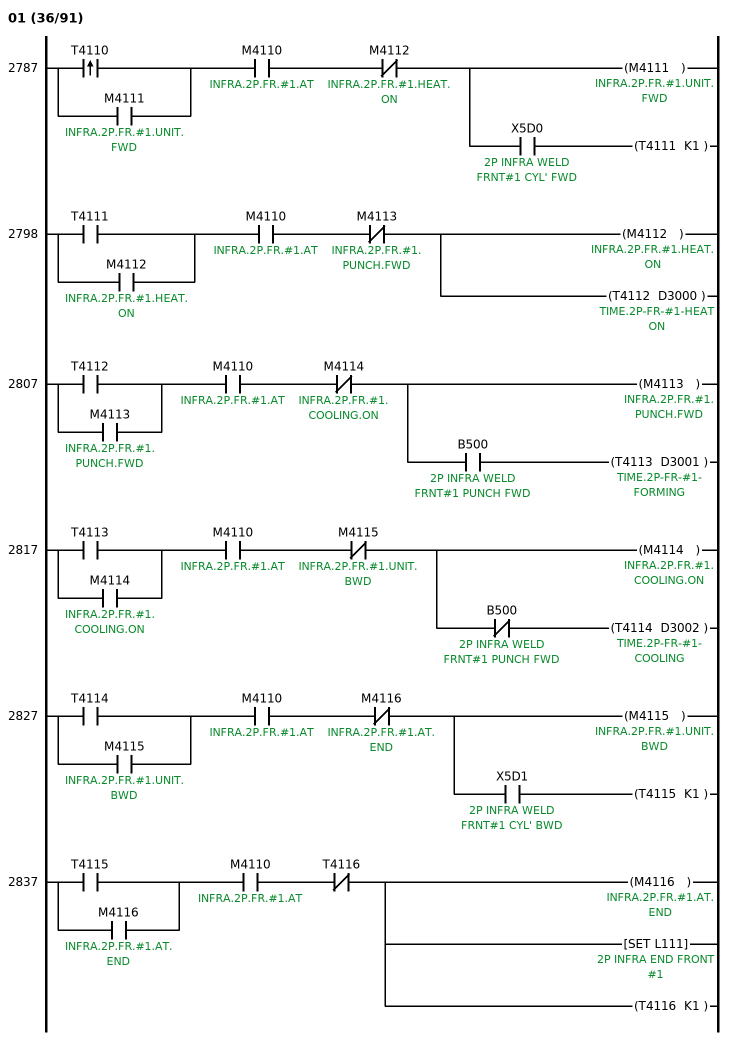
2787  LDP     T4110
      OR      M4111  ; INFRA.2P.FR.#1.UNIT.FWD
      AND     M4110  ; INFRA.2P.FR.#1.AT
      ANI     M4112  ; INFRA.2P.FR.#1.HEAT.ON
      OUT     M4111  ; INFRA.2P.FR.#1.UNIT.FWD
      AND     X5D0  ; 2P INFRA WELD FRNT#1 CYL' FWD
      OUT     T4111 K1
2798  LD      T4111
      OR      M4112  ; INFRA.2P.FR.#1.HEAT.ON
      AND     M4110  ; INFRA.2P.FR.#1.AT
      ANI     M4113  ; INFRA.2P.FR.#1.PUNCH.FWD
      OUT     M4112  ; INFRA.2P.FR.#1.HEAT.ON
      OUT     T4112 D3000  ; TIME.2P-FR-#1-HEAT ON
2807  LD      T4112
      OR      M4113  ; INFRA.2P.FR.#1.PUNCH.FWD
      AND     M4110  ; INFRA.2P.FR.#1.AT
      ANI     M4114  ; INFRA.2P.FR.#1.COOLING.ON
      OUT     M4113  ; INFRA.2P.FR.#1.PUNCH.FWD
      AND     B500  ; 2P INFRA WELD FRNT#1 PUNCH FWD
      OUT     T4113 D3001  ; TIME.2P-FR-#1-FORMING
2817  LD      T4113
      OR      M4114  ; INFRA.2P.FR.#1.COOLING.ON
      AND     M4110  ; INFRA.2P.FR.#1.AT
      ANI     M4115  ; INFRA.2P.FR.#1.UNIT.BWD
      OUT     M4114  ; INFRA.2P.FR.#1.COOLING.ON
      ANI     B500  ; 2P INFRA WELD FRNT#1 PUNCH FWD
      OUT     T4114 D3002  ; TIME.2P-FR-#1-COOLING
2827  LD      T4114
      OR      M4115  ; INFRA.2P.FR.#1.UNIT.BWD
      AND     M4110  ; INFRA.2P.FR.#1.AT
      ANI     M4116  ; INFRA.2P.FR.#1.AT.END
      OUT     M4115  ; INFRA.2P.FR.#1.UNIT.BWD
      AND     X5D1  ; 2P INFRA WELD FRNT#1 CYL' BWD
      OUT     T4115 K1
2837  LD      T4115
      OR      M4116  ; INFRA.2P.FR.#1.AT.END
      AND     M4110  ; INFRA.2P.FR.#1.AT
      ANI     T4116
      OUT     M4116  ; INFRA.2P.FR.#1.AT.END
      SET     L111  ; 2P INFRA END FRONT #1
      OUT     T4116 K1
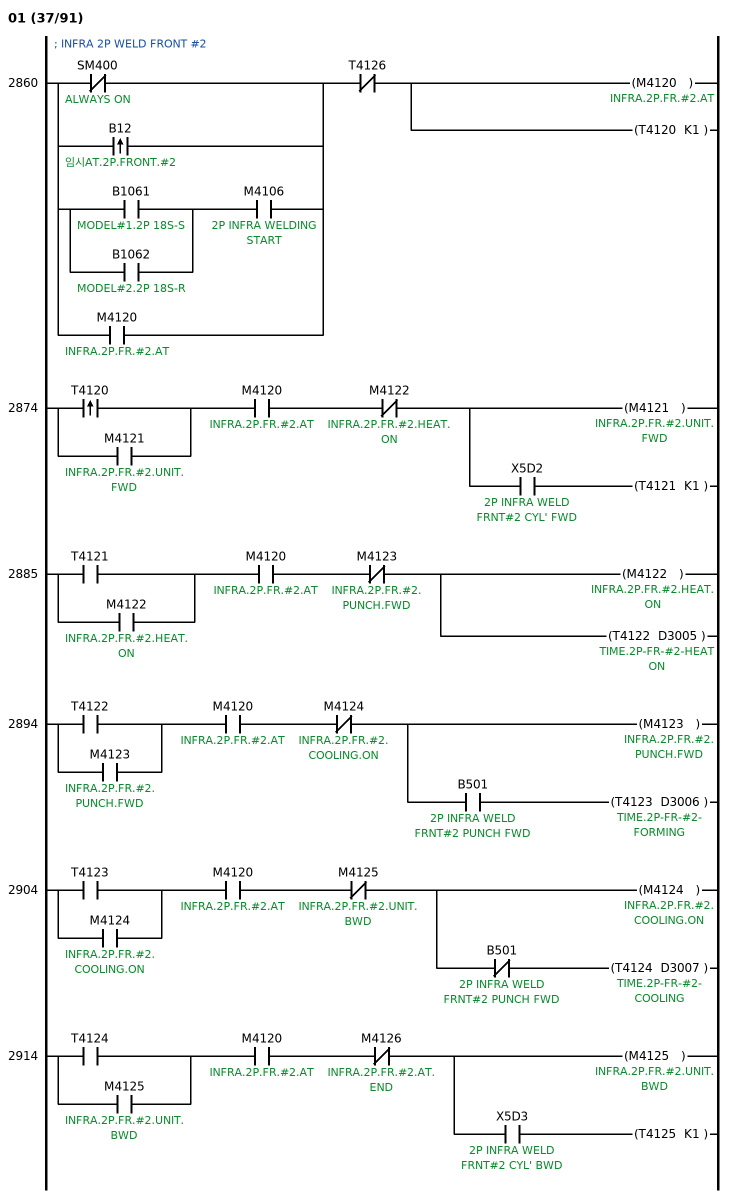
; INFRA 2P WELD FRONT #2
2860  LDI     SM400  ; ALWAYS ON
      ORP     B12  ; 임시AT.2P.FRONT.#2
      LD      B1061  ; MODEL#1.2P 18S-S
      OR      B1062  ; MODEL#2.2P 18S-R
      AND     M4106  ; 2P INFRA WELDING START
      ORB
      OR      M4120  ; INFRA.2P.FR.#2.AT
      ANI     T4126
      OUT     M4120  ; INFRA.2P.FR.#2.AT
      OUT     T4120 K1
2874  LDP     T4120
      OR      M4121  ; INFRA.2P.FR.#2.UNIT.FWD
      AND     M4120  ; INFRA.2P.FR.#2.AT
      ANI     M4122  ; INFRA.2P.FR.#2.HEAT.ON
      OUT     M4121  ; INFRA.2P.FR.#2.UNIT.FWD
      AND     X5D2  ; 2P INFRA WELD FRNT#2 CYL' FWD
      OUT     T4121 K1
2885  LD      T4121
      OR      M4122  ; INFRA.2P.FR.#2.HEAT.ON
      AND     M4120  ; INFRA.2P.FR.#2.AT
      ANI     M4123  ; INFRA.2P.FR.#2.PUNCH.FWD
      OUT     M4122  ; INFRA.2P.FR.#2.HEAT.ON
      OUT     T4122 D3005  ; TIME.2P-FR-#2-HEAT ON
2894  LD      T4122
      OR      M4123  ; INFRA.2P.FR.#2.PUNCH.FWD
      AND     M4120  ; INFRA.2P.FR.#2.AT
      ANI     M4124  ; INFRA.2P.FR.#2.COOLING.ON
      OUT     M4123  ; INFRA.2P.FR.#2.PUNCH.FWD
      AND     B501  ; 2P INFRA WELD FRNT#2 PUNCH FWD
      OUT     T4123 D3006  ; TIME.2P-FR-#2-FORMING
2904  LD      T4123
      OR      M4124  ; INFRA.2P.FR.#2.COOLING.ON
      AND     M4120  ; INFRA.2P.FR.#2.AT
      ANI     M4125  ; INFRA.2P.FR.#2.UNIT.BWD
      OUT     M4124  ; INFRA.2P.FR.#2.COOLING.ON
      ANI     B501  ; 2P INFRA WELD FRNT#2 PUNCH FWD
      OUT     T4124 D3007  ; TIME.2P-FR-#2-COOLING
2914  LD      T4124
      OR      M4125  ; INFRA.2P.FR.#2.UNIT.BWD
      AND     M4120  ; INFRA.2P.FR.#2.AT
      ANI     M4126  ; INFRA.2P.FR.#2.AT.END
      OUT     M4125  ; INFRA.2P.FR.#2.UNIT.BWD
      AND     X5D3  ; 2P INFRA WELD FRNT#2 CYL' BWD
      OUT     T4125 K1
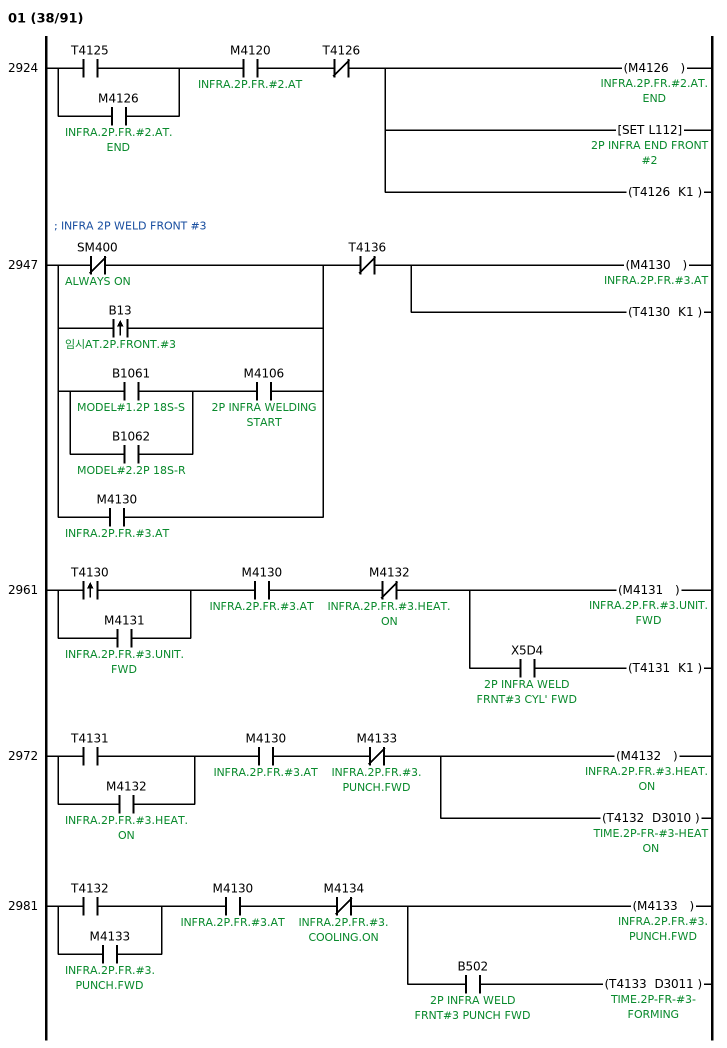
2924  LD      T4125
      OR      M4126  ; INFRA.2P.FR.#2.AT.END
      AND     M4120  ; INFRA.2P.FR.#2.AT
      ANI     T4126
      OUT     M4126  ; INFRA.2P.FR.#2.AT.END
      SET     L112  ; 2P INFRA END FRONT #2
      OUT     T4126 K1
; INFRA 2P WELD FRONT #3
2947  LDI     SM400  ; ALWAYS ON
      ORP     B13  ; 임시AT.2P.FRONT.#3
      LD      B1061  ; MODEL#1.2P 18S-S
      OR      B1062  ; MODEL#2.2P 18S-R
      AND     M4106  ; 2P INFRA WELDING START
      ORB
      OR      M4130  ; INFRA.2P.FR.#3.AT
      ANI     T4136
      OUT     M4130  ; INFRA.2P.FR.#3.AT
      OUT     T4130 K1
2961  LDP     T4130
      OR      M4131  ; INFRA.2P.FR.#3.UNIT.FWD
      AND     M4130  ; INFRA.2P.FR.#3.AT
      ANI     M4132  ; INFRA.2P.FR.#3.HEAT.ON
      OUT     M4131  ; INFRA.2P.FR.#3.UNIT.FWD
      AND     X5D4  ; 2P INFRA WELD FRNT#3 CYL' FWD
      OUT     T4131 K1
2972  LD      T4131
      OR      M4132  ; INFRA.2P.FR.#3.HEAT.ON
      AND     M4130  ; INFRA.2P.FR.#3.AT
      ANI     M4133  ; INFRA.2P.FR.#3.PUNCH.FWD
      OUT     M4132  ; INFRA.2P.FR.#3.HEAT.ON
      OUT     T4132 D3010  ; TIME.2P-FR-#3-HEAT ON
2981  LD      T4132
      OR      M4133  ; INFRA.2P.FR.#3.PUNCH.FWD
      AND     M4130  ; INFRA.2P.FR.#3.AT
      ANI     M4134  ; INFRA.2P.FR.#3.COOLING.ON
      OUT     M4133  ; INFRA.2P.FR.#3.PUNCH.FWD
      AND     B502  ; 2P INFRA WELD FRNT#3 PUNCH FWD
      OUT     T4133 D3011  ; TIME.2P-FR-#3-FORMING
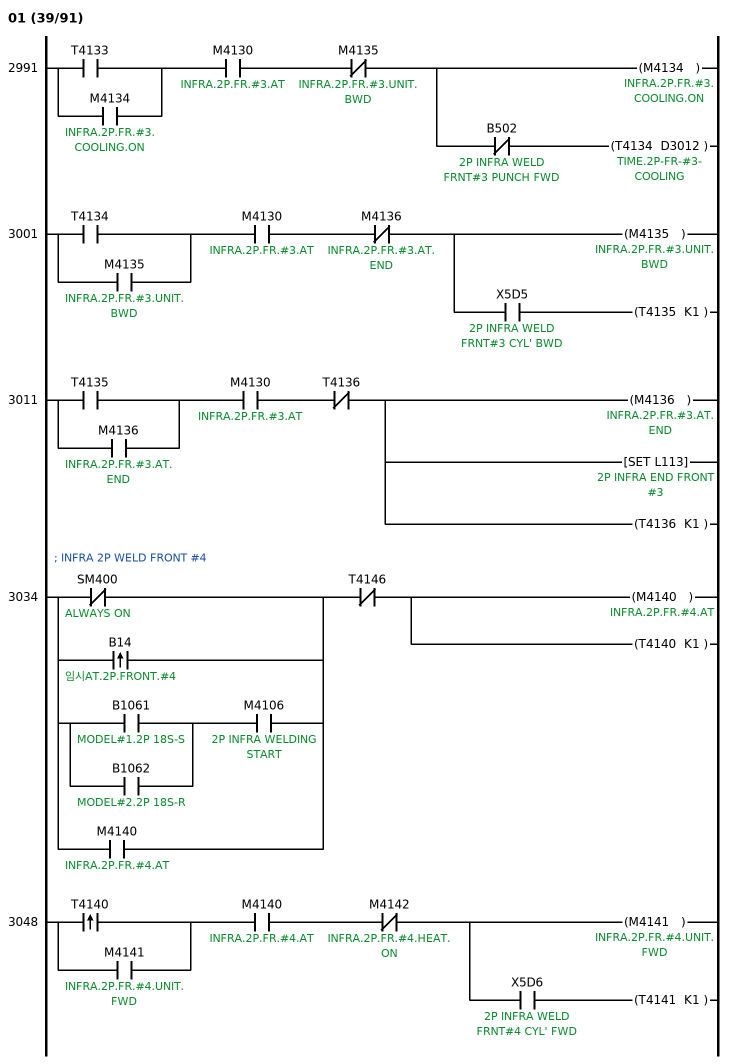
2991  LD      T4133
      OR      M4134  ; INFRA.2P.FR.#3.COOLING.ON
      AND     M4130  ; INFRA.2P.FR.#3.AT
      ANI     M4135  ; INFRA.2P.FR.#3.UNIT.BWD
      OUT     M4134  ; INFRA.2P.FR.#3.COOLING.ON
      ANI     B502  ; 2P INFRA WELD FRNT#3 PUNCH FWD
      OUT     T4134 D3012  ; TIME.2P-FR-#3-COOLING
3001  LD      T4134
      OR      M4135  ; INFRA.2P.FR.#3.UNIT.BWD
      AND     M4130  ; INFRA.2P.FR.#3.AT
      ANI     M4136  ; INFRA.2P.FR.#3.AT.END
      OUT     M4135  ; INFRA.2P.FR.#3.UNIT.BWD
      AND     X5D5  ; 2P INFRA WELD FRNT#3 CYL' BWD
      OUT     T4135 K1
3011  LD      T4135
      OR      M4136  ; INFRA.2P.FR.#3.AT.END
      AND     M4130  ; INFRA.2P.FR.#3.AT
      ANI     T4136
      OUT     M4136  ; INFRA.2P.FR.#3.AT.END
      SET     L113  ; 2P INFRA END FRONT #3
      OUT     T4136 K1
; INFRA 2P WELD FRONT #4
3034  LDI     SM400  ; ALWAYS ON
      ORP     B14  ; 임시AT.2P.FRONT.#4
      LD      B1061  ; MODEL#1.2P 18S-S
      OR      B1062  ; MODEL#2.2P 18S-R
      AND     M4106  ; 2P INFRA WELDING START
      ORB
      OR      M4140  ; INFRA.2P.FR.#4.AT
      ANI     T4146
      OUT     M4140  ; INFRA.2P.FR.#4.AT
      OUT     T4140 K1
3048  LDP     T4140
      OR      M4141  ; INFRA.2P.FR.#4.UNIT.FWD
      AND     M4140  ; INFRA.2P.FR.#4.AT
      ANI     M4142  ; INFRA.2P.FR.#4.HEAT.ON
      OUT     M4141  ; INFRA.2P.FR.#4.UNIT.FWD
      AND     X5D6  ; 2P INFRA WELD FRNT#4 CYL' FWD
      OUT     T4141 K1
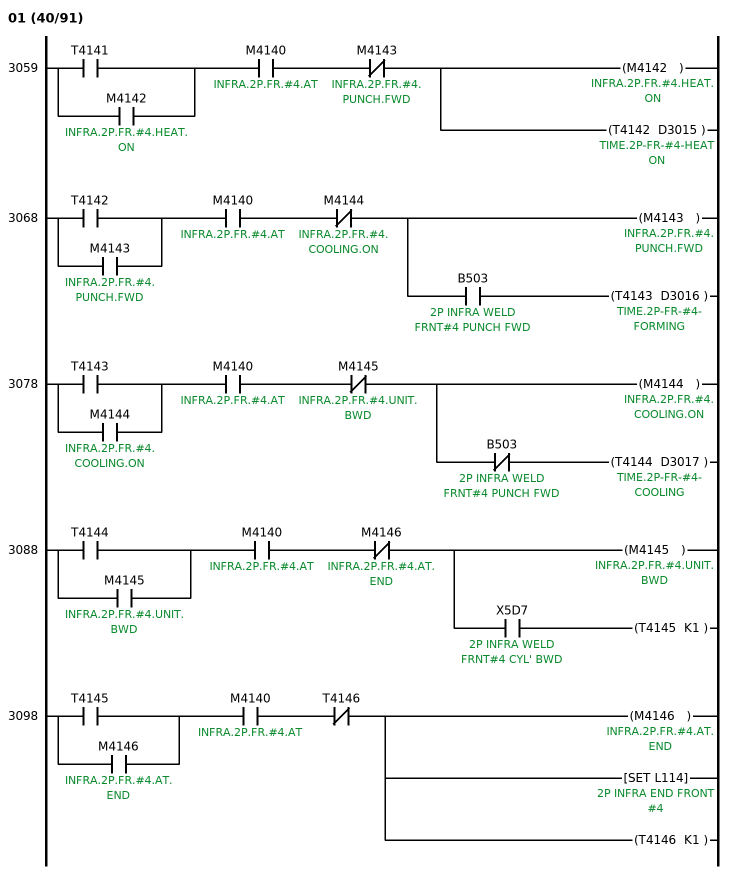
3059  LD      T4141
      OR      M4142  ; INFRA.2P.FR.#4.HEAT.ON
      AND     M4140  ; INFRA.2P.FR.#4.AT
      ANI     M4143  ; INFRA.2P.FR.#4.PUNCH.FWD
      OUT     M4142  ; INFRA.2P.FR.#4.HEAT.ON
      OUT     T4142 D3015  ; TIME.2P-FR-#4-HEAT ON
3068  LD      T4142
      OR      M4143  ; INFRA.2P.FR.#4.PUNCH.FWD
      AND     M4140  ; INFRA.2P.FR.#4.AT
      ANI     M4144  ; INFRA.2P.FR.#4.COOLING.ON
      OUT     M4143  ; INFRA.2P.FR.#4.PUNCH.FWD
      AND     B503  ; 2P INFRA WELD FRNT#4 PUNCH FWD
      OUT     T4143 D3016  ; TIME.2P-FR-#4-FORMING
3078  LD      T4143
      OR      M4144  ; INFRA.2P.FR.#4.COOLING.ON
      AND     M4140  ; INFRA.2P.FR.#4.AT
      ANI     M4145  ; INFRA.2P.FR.#4.UNIT.BWD
      OUT     M4144  ; INFRA.2P.FR.#4.COOLING.ON
      ANI     B503  ; 2P INFRA WELD FRNT#4 PUNCH FWD
      OUT     T4144 D3017  ; TIME.2P-FR-#4-COOLING
3088  LD      T4144
      OR      M4145  ; INFRA.2P.FR.#4.UNIT.BWD
      AND     M4140  ; INFRA.2P.FR.#4.AT
      ANI     M4146  ; INFRA.2P.FR.#4.AT.END
      OUT     M4145  ; INFRA.2P.FR.#4.UNIT.BWD
      AND     X5D7  ; 2P INFRA WELD FRNT#4 CYL' BWD
      OUT     T4145 K1
3098  LD      T4145
      OR      M4146  ; INFRA.2P.FR.#4.AT.END
      AND     M4140  ; INFRA.2P.FR.#4.AT
      ANI     T4146
      OUT     M4146  ; INFRA.2P.FR.#4.AT.END
      SET     L114  ; 2P INFRA END FRONT #4
      OUT     T4146 K1
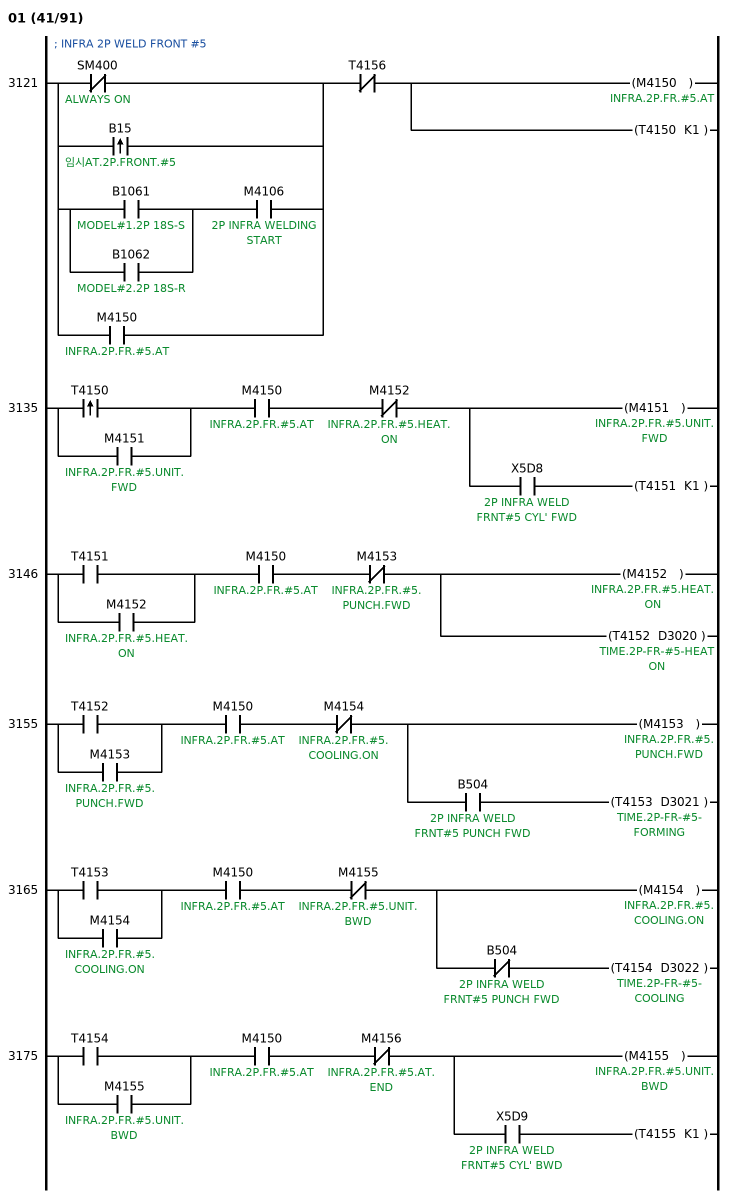
; INFRA 2P WELD FRONT #5
3121  LDI     SM400  ; ALWAYS ON
      ORP     B15  ; 임시AT.2P.FRONT.#5
      LD      B1061  ; MODEL#1.2P 18S-S
      OR      B1062  ; MODEL#2.2P 18S-R
      AND     M4106  ; 2P INFRA WELDING START
      ORB
      OR      M4150  ; INFRA.2P.FR.#5.AT
      ANI     T4156
      OUT     M4150  ; INFRA.2P.FR.#5.AT
      OUT     T4150 K1
3135  LDP     T4150
      OR      M4151  ; INFRA.2P.FR.#5.UNIT.FWD
      AND     M4150  ; INFRA.2P.FR.#5.AT
      ANI     M4152  ; INFRA.2P.FR.#5.HEAT.ON
      OUT     M4151  ; INFRA.2P.FR.#5.UNIT.FWD
      AND     X5D8  ; 2P INFRA WELD FRNT#5 CYL' FWD
      OUT     T4151 K1
3146  LD      T4151
      OR      M4152  ; INFRA.2P.FR.#5.HEAT.ON
      AND     M4150  ; INFRA.2P.FR.#5.AT
      ANI     M4153  ; INFRA.2P.FR.#5.PUNCH.FWD
      OUT     M4152  ; INFRA.2P.FR.#5.HEAT.ON
      OUT     T4152 D3020  ; TIME.2P-FR-#5-HEAT ON
3155  LD      T4152
      OR      M4153  ; INFRA.2P.FR.#5.PUNCH.FWD
      AND     M4150  ; INFRA.2P.FR.#5.AT
      ANI     M4154  ; INFRA.2P.FR.#5.COOLING.ON
      OUT     M4153  ; INFRA.2P.FR.#5.PUNCH.FWD
      AND     B504  ; 2P INFRA WELD FRNT#5 PUNCH FWD
      OUT     T4153 D3021  ; TIME.2P-FR-#5-FORMING
3165  LD      T4153
      OR      M4154  ; INFRA.2P.FR.#5.COOLING.ON
      AND     M4150  ; INFRA.2P.FR.#5.AT
      ANI     M4155  ; INFRA.2P.FR.#5.UNIT.BWD
      OUT     M4154  ; INFRA.2P.FR.#5.COOLING.ON
      ANI     B504  ; 2P INFRA WELD FRNT#5 PUNCH FWD
      OUT     T4154 D3022  ; TIME.2P-FR-#5-COOLING
3175  LD      T4154
      OR      M4155  ; INFRA.2P.FR.#5.UNIT.BWD
      AND     M4150  ; INFRA.2P.FR.#5.AT
      ANI     M4156  ; INFRA.2P.FR.#5.AT.END
      OUT     M4155  ; INFRA.2P.FR.#5.UNIT.BWD
      AND     X5D9  ; 2P INFRA WELD FRNT#5 CYL' BWD
      OUT     T4155 K1
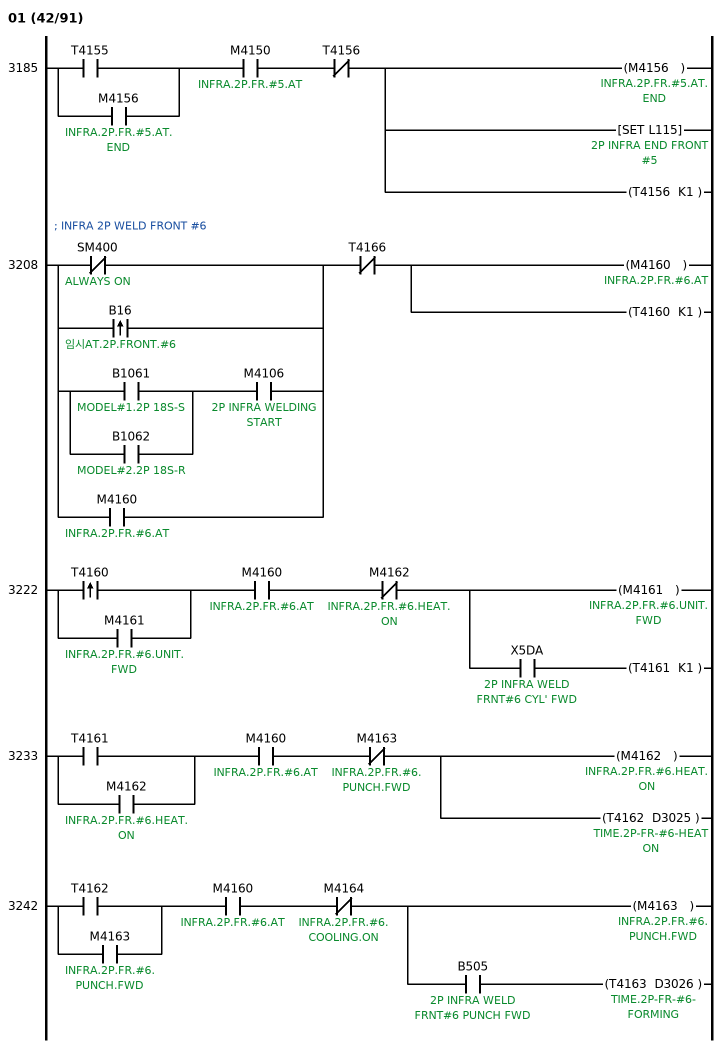
3185  LD      T4155
      OR      M4156  ; INFRA.2P.FR.#5.AT.END
      AND     M4150  ; INFRA.2P.FR.#5.AT
      ANI     T4156
      OUT     M4156  ; INFRA.2P.FR.#5.AT.END
      SET     L115  ; 2P INFRA END FRONT #5
      OUT     T4156 K1
; INFRA 2P WELD FRONT #6
3208  LDI     SM400  ; ALWAYS ON
      ORP     B16  ; 임시AT.2P.FRONT.#6
      LD      B1061  ; MODEL#1.2P 18S-S
      OR      B1062  ; MODEL#2.2P 18S-R
      AND     M4106  ; 2P INFRA WELDING START
      ORB
      OR      M4160  ; INFRA.2P.FR.#6.AT
      ANI     T4166
      OUT     M4160  ; INFRA.2P.FR.#6.AT
      OUT     T4160 K1
3222  LDP     T4160
      OR      M4161  ; INFRA.2P.FR.#6.UNIT.FWD
      AND     M4160  ; INFRA.2P.FR.#6.AT
      ANI     M4162  ; INFRA.2P.FR.#6.HEAT.ON
      OUT     M4161  ; INFRA.2P.FR.#6.UNIT.FWD
      AND     X5DA  ; 2P INFRA WELD FRNT#6 CYL' FWD
      OUT     T4161 K1
3233  LD      T4161
      OR      M4162  ; INFRA.2P.FR.#6.HEAT.ON
      AND     M4160  ; INFRA.2P.FR.#6.AT
      ANI     M4163  ; INFRA.2P.FR.#6.PUNCH.FWD
      OUT     M4162  ; INFRA.2P.FR.#6.HEAT.ON
      OUT     T4162 D3025  ; TIME.2P-FR-#6-HEAT ON
3242  LD      T4162
      OR      M4163  ; INFRA.2P.FR.#6.PUNCH.FWD
      AND     M4160  ; INFRA.2P.FR.#6.AT
      ANI     M4164  ; INFRA.2P.FR.#6.COOLING.ON
      OUT     M4163  ; INFRA.2P.FR.#6.PUNCH.FWD
      AND     B505  ; 2P INFRA WELD FRNT#6 PUNCH FWD
      OUT     T4163 D3026  ; TIME.2P-FR-#6-FORMING
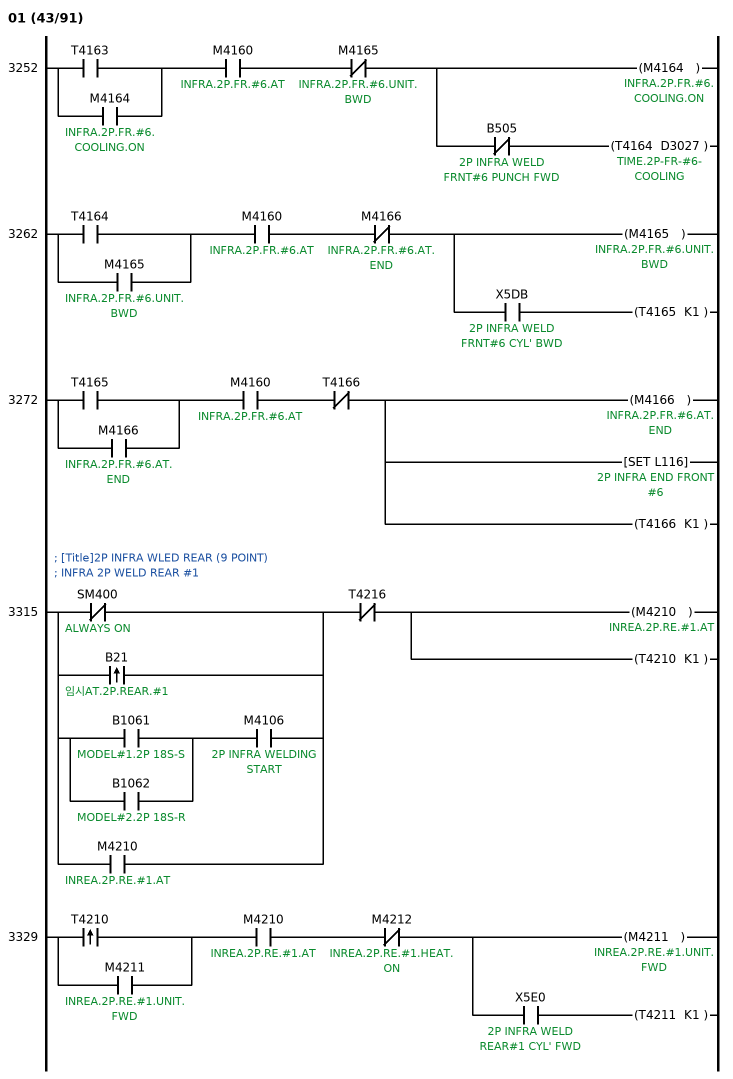
3252  LD      T4163
      OR      M4164  ; INFRA.2P.FR.#6.COOLING.ON
      AND     M4160  ; INFRA.2P.FR.#6.AT
      ANI     M4165  ; INFRA.2P.FR.#6.UNIT.BWD
      OUT     M4164  ; INFRA.2P.FR.#6.COOLING.ON
      ANI     B505  ; 2P INFRA WELD FRNT#6 PUNCH FWD
      OUT     T4164 D3027  ; TIME.2P-FR-#6-COOLING
3262  LD      T4164
      OR      M4165  ; INFRA.2P.FR.#6.UNIT.BWD
      AND     M4160  ; INFRA.2P.FR.#6.AT
      ANI     M4166  ; INFRA.2P.FR.#6.AT.END
      OUT     M4165  ; INFRA.2P.FR.#6.UNIT.BWD
      AND     X5DB  ; 2P INFRA WELD FRNT#6 CYL' BWD
      OUT     T4165 K1
3272  LD      T4165
      OR      M4166  ; INFRA.2P.FR.#6.AT.END
      AND     M4160  ; INFRA.2P.FR.#6.AT
      ANI     T4166
      OUT     M4166  ; INFRA.2P.FR.#6.AT.END
      SET     L116  ; 2P INFRA END FRONT #6
      OUT     T4166 K1
; [Title]2P INFRA WLED REAR (9 POINT)
; INFRA 2P WELD REAR #1
3315  LDI     SM400  ; ALWAYS ON
      ORP     B21  ; 임시AT.2P.REAR.#1
      LD      B1061  ; MODEL#1.2P 18S-S
      OR      B1062  ; MODEL#2.2P 18S-R
      AND     M4106  ; 2P INFRA WELDING START
      ORB
      OR      M4210  ; INREA.2P.RE.#1.AT
      ANI     T4216
      OUT     M4210  ; INREA.2P.RE.#1.AT
      OUT     T4210 K1
3329  LDP     T4210
      OR      M4211  ; INREA.2P.RE.#1.UNIT.FWD
      AND     M4210  ; INREA.2P.RE.#1.AT
      ANI     M4212  ; INREA.2P.RE.#1.HEAT.ON
      OUT     M4211  ; INREA.2P.RE.#1.UNIT.FWD
      AND     X5E0  ; 2P INFRA WELD REAR#1 CYL' FWD
      OUT     T4211 K1
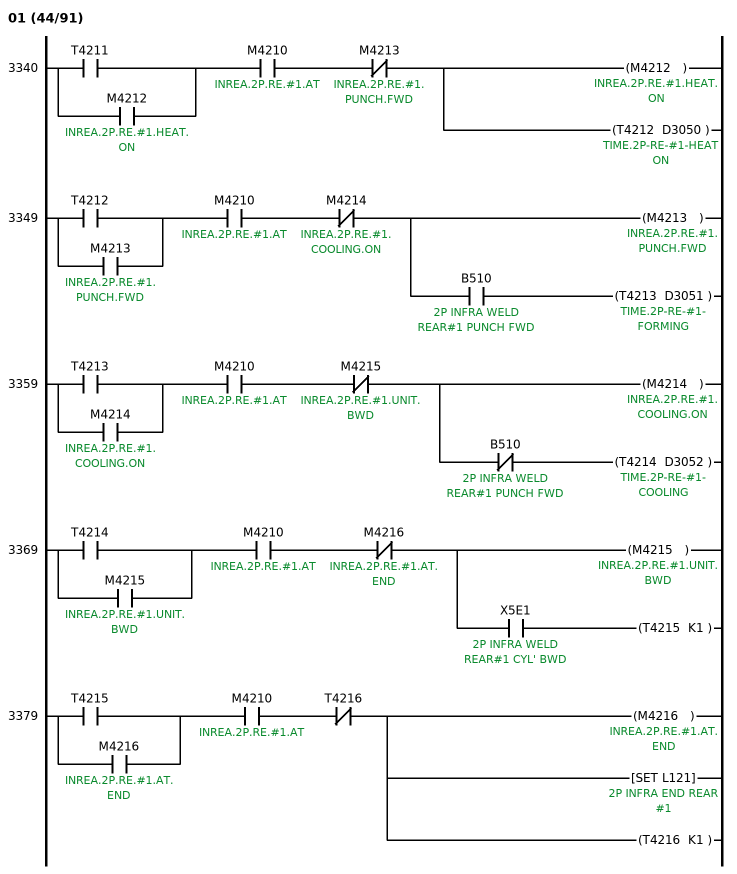
3340  LD      T4211
      OR      M4212  ; INREA.2P.RE.#1.HEAT.ON
      AND     M4210  ; INREA.2P.RE.#1.AT
      ANI     M4213  ; INREA.2P.RE.#1.PUNCH.FWD
      OUT     M4212  ; INREA.2P.RE.#1.HEAT.ON
      OUT     T4212 D3050  ; TIME.2P-RE-#1-HEAT ON
3349  LD      T4212
      OR      M4213  ; INREA.2P.RE.#1.PUNCH.FWD
      AND     M4210  ; INREA.2P.RE.#1.AT
      ANI     M4214  ; INREA.2P.RE.#1.COOLING.ON
      OUT     M4213  ; INREA.2P.RE.#1.PUNCH.FWD
      AND     B510  ; 2P INFRA WELD REAR#1 PUNCH FWD
      OUT     T4213 D3051  ; TIME.2P-RE-#1-FORMING
3359  LD      T4213
      OR      M4214  ; INREA.2P.RE.#1.COOLING.ON
      AND     M4210  ; INREA.2P.RE.#1.AT
      ANI     M4215  ; INREA.2P.RE.#1.UNIT.BWD
      OUT     M4214  ; INREA.2P.RE.#1.COOLING.ON
      ANI     B510  ; 2P INFRA WELD REAR#1 PUNCH FWD
      OUT     T4214 D3052  ; TIME.2P-RE-#1-COOLING
3369  LD      T4214
      OR      M4215  ; INREA.2P.RE.#1.UNIT.BWD
      AND     M4210  ; INREA.2P.RE.#1.AT
      ANI     M4216  ; INREA.2P.RE.#1.AT.END
      OUT     M4215  ; INREA.2P.RE.#1.UNIT.BWD
      AND     X5E1  ; 2P INFRA WELD REAR#1 CYL' BWD
      OUT     T4215 K1
3379  LD      T4215
      OR      M4216  ; INREA.2P.RE.#1.AT.END
      AND     M4210  ; INREA.2P.RE.#1.AT
      ANI     T4216
      OUT     M4216  ; INREA.2P.RE.#1.AT.END
      SET     L121  ; 2P INFRA END REAR #1
      OUT     T4216 K1
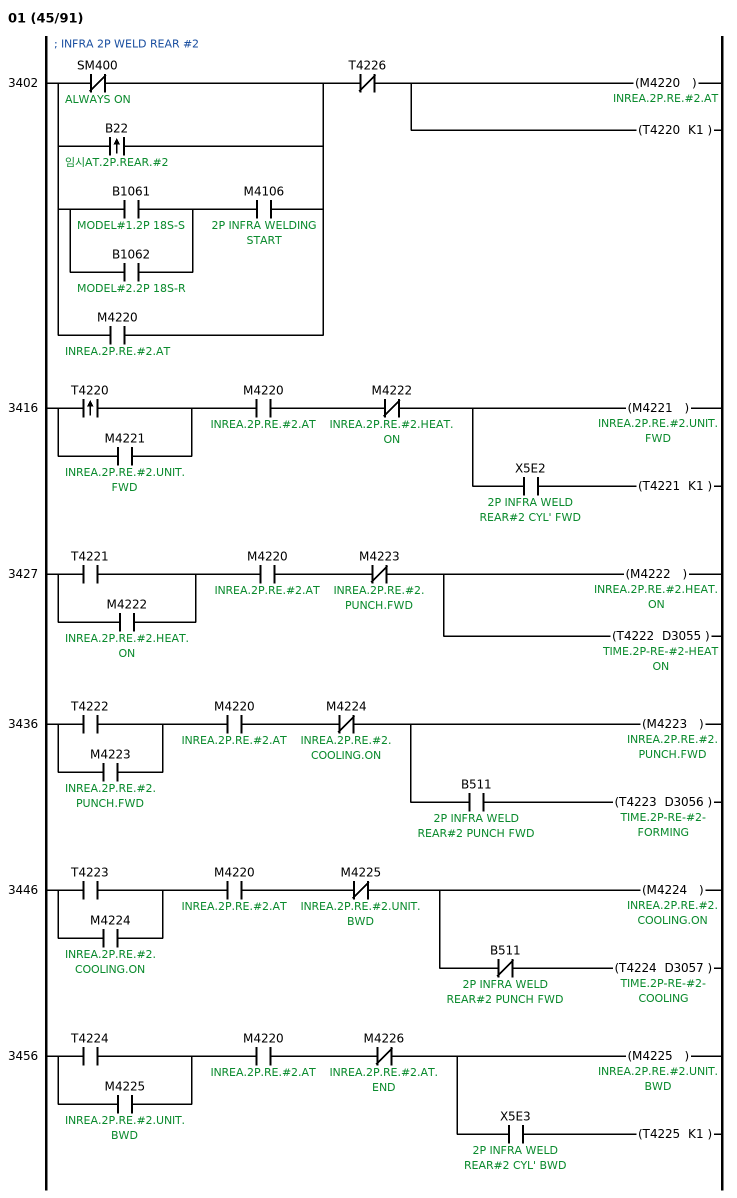
; INFRA 2P WELD REAR #2
3402  LDI     SM400  ; ALWAYS ON
      ORP     B22  ; 임시AT.2P.REAR.#2
      LD      B1061  ; MODEL#1.2P 18S-S
      OR      B1062  ; MODEL#2.2P 18S-R
      AND     M4106  ; 2P INFRA WELDING START
      ORB
      OR      M4220  ; INREA.2P.RE.#2.AT
      ANI     T4226
      OUT     M4220  ; INREA.2P.RE.#2.AT
      OUT     T4220 K1
3416  LDP     T4220
      OR      M4221  ; INREA.2P.RE.#2.UNIT.FWD
      AND     M4220  ; INREA.2P.RE.#2.AT
      ANI     M4222  ; INREA.2P.RE.#2.HEAT.ON
      OUT     M4221  ; INREA.2P.RE.#2.UNIT.FWD
      AND     X5E2  ; 2P INFRA WELD REAR#2 CYL' FWD
      OUT     T4221 K1
3427  LD      T4221
      OR      M4222  ; INREA.2P.RE.#2.HEAT.ON
      AND     M4220  ; INREA.2P.RE.#2.AT
      ANI     M4223  ; INREA.2P.RE.#2.PUNCH.FWD
      OUT     M4222  ; INREA.2P.RE.#2.HEAT.ON
      OUT     T4222 D3055  ; TIME.2P-RE-#2-HEAT ON
3436  LD      T4222
      OR      M4223  ; INREA.2P.RE.#2.PUNCH.FWD
      AND     M4220  ; INREA.2P.RE.#2.AT
      ANI     M4224  ; INREA.2P.RE.#2.COOLING.ON
      OUT     M4223  ; INREA.2P.RE.#2.PUNCH.FWD
      AND     B511  ; 2P INFRA WELD REAR#2 PUNCH FWD
      OUT     T4223 D3056  ; TIME.2P-RE-#2-FORMING
3446  LD      T4223
      OR      M4224  ; INREA.2P.RE.#2.COOLING.ON
      AND     M4220  ; INREA.2P.RE.#2.AT
      ANI     M4225  ; INREA.2P.RE.#2.UNIT.BWD
      OUT     M4224  ; INREA.2P.RE.#2.COOLING.ON
      ANI     B511  ; 2P INFRA WELD REAR#2 PUNCH FWD
      OUT     T4224 D3057  ; TIME.2P-RE-#2-COOLING
3456  LD      T4224
      OR      M4225  ; INREA.2P.RE.#2.UNIT.BWD
      AND     M4220  ; INREA.2P.RE.#2.AT
      ANI     M4226  ; INREA.2P.RE.#2.AT.END
      OUT     M4225  ; INREA.2P.RE.#2.UNIT.BWD
      AND     X5E3  ; 2P INFRA WELD REAR#2 CYL' BWD
      OUT     T4225 K1
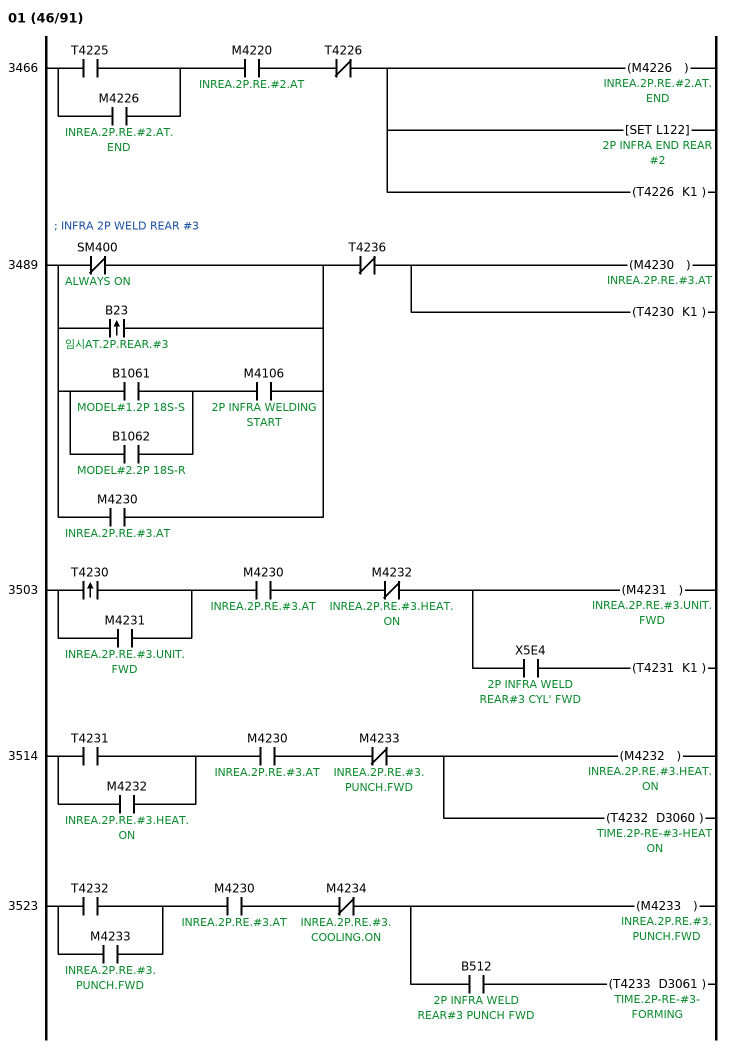
3466  LD      T4225
      OR      M4226  ; INREA.2P.RE.#2.AT.END
      AND     M4220  ; INREA.2P.RE.#2.AT
      ANI     T4226
      OUT     M4226  ; INREA.2P.RE.#2.AT.END
      SET     L122  ; 2P INFRA END REAR #2
      OUT     T4226 K1
; INFRA 2P WELD REAR #3
3489  LDI     SM400  ; ALWAYS ON
      ORP     B23  ; 임시AT.2P.REAR.#3
      LD      B1061  ; MODEL#1.2P 18S-S
      OR      B1062  ; MODEL#2.2P 18S-R
      AND     M4106  ; 2P INFRA WELDING START
      ORB
      OR      M4230  ; INREA.2P.RE.#3.AT
      ANI     T4236
      OUT     M4230  ; INREA.2P.RE.#3.AT
      OUT     T4230 K1
3503  LDP     T4230
      OR      M4231  ; INREA.2P.RE.#3.UNIT.FWD
      AND     M4230  ; INREA.2P.RE.#3.AT
      ANI     M4232  ; INREA.2P.RE.#3.HEAT.ON
      OUT     M4231  ; INREA.2P.RE.#3.UNIT.FWD
      AND     X5E4  ; 2P INFRA WELD REAR#3 CYL' FWD
      OUT     T4231 K1
3514  LD      T4231
      OR      M4232  ; INREA.2P.RE.#3.HEAT.ON
      AND     M4230  ; INREA.2P.RE.#3.AT
      ANI     M4233  ; INREA.2P.RE.#3.PUNCH.FWD
      OUT     M4232  ; INREA.2P.RE.#3.HEAT.ON
      OUT     T4232 D3060  ; TIME.2P-RE-#3-HEAT ON
3523  LD      T4232
      OR      M4233  ; INREA.2P.RE.#3.PUNCH.FWD
      AND     M4230  ; INREA.2P.RE.#3.AT
      ANI     M4234  ; INREA.2P.RE.#3.COOLING.ON
      OUT     M4233  ; INREA.2P.RE.#3.PUNCH.FWD
      AND     B512  ; 2P INFRA WELD REAR#3 PUNCH FWD
      OUT     T4233 D3061  ; TIME.2P-RE-#3-FORMING
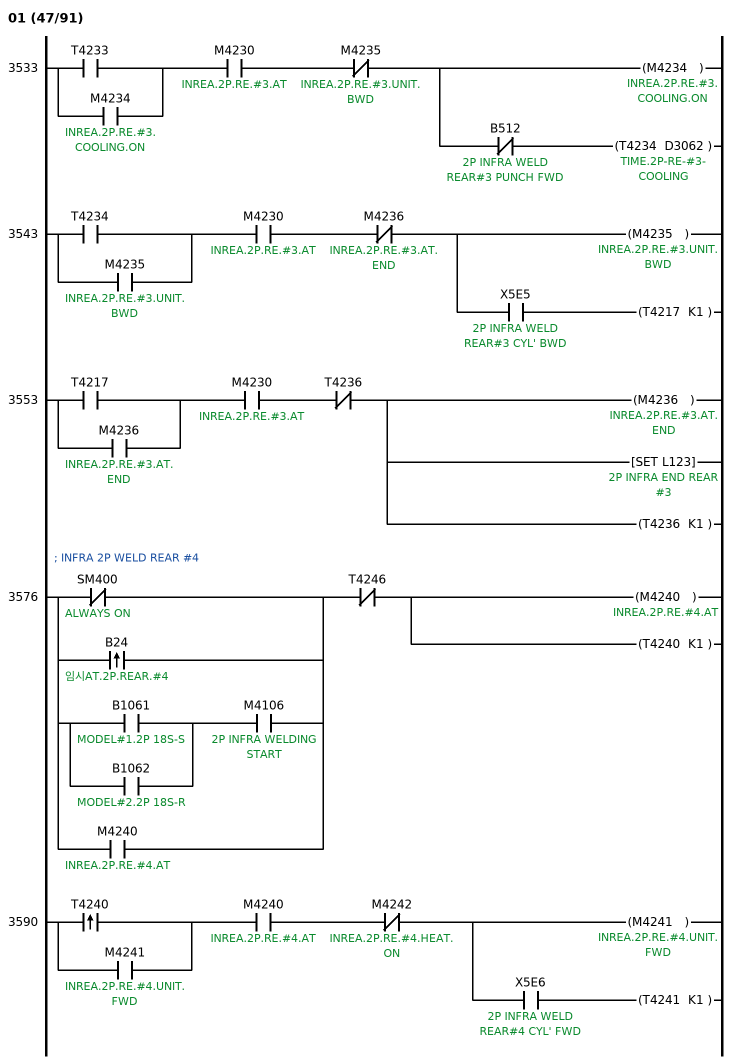
3533  LD      T4233
      OR      M4234  ; INREA.2P.RE.#3.COOLING.ON
      AND     M4230  ; INREA.2P.RE.#3.AT
      ANI     M4235  ; INREA.2P.RE.#3.UNIT.BWD
      OUT     M4234  ; INREA.2P.RE.#3.COOLING.ON
      ANI     B512  ; 2P INFRA WELD REAR#3 PUNCH FWD
      OUT     T4234 D3062  ; TIME.2P-RE-#3-COOLING
3543  LD      T4234
      OR      M4235  ; INREA.2P.RE.#3.UNIT.BWD
      AND     M4230  ; INREA.2P.RE.#3.AT
      ANI     M4236  ; INREA.2P.RE.#3.AT.END
      OUT     M4235  ; INREA.2P.RE.#3.UNIT.BWD
      AND     X5E5  ; 2P INFRA WELD REAR#3 CYL' BWD
      OUT     T4217 K1
3553  LD      T4217
      OR      M4236  ; INREA.2P.RE.#3.AT.END
      AND     M4230  ; INREA.2P.RE.#3.AT
      ANI     T4236
      OUT     M4236  ; INREA.2P.RE.#3.AT.END
      SET     L123  ; 2P INFRA END REAR #3
      OUT     T4236 K1
; INFRA 2P WELD REAR #4
3576  LDI     SM400  ; ALWAYS ON
      ORP     B24  ; 임시AT.2P.REAR.#4
      LD      B1061  ; MODEL#1.2P 18S-S
      OR      B1062  ; MODEL#2.2P 18S-R
      AND     M4106  ; 2P INFRA WELDING START
      ORB
      OR      M4240  ; INREA.2P.RE.#4.AT
      ANI     T4246
      OUT     M4240  ; INREA.2P.RE.#4.AT
      OUT     T4240 K1
3590  LDP     T4240
      OR      M4241  ; INREA.2P.RE.#4.UNIT.FWD
      AND     M4240  ; INREA.2P.RE.#4.AT
      ANI     M4242  ; INREA.2P.RE.#4.HEAT.ON
      OUT     M4241  ; INREA.2P.RE.#4.UNIT.FWD
      AND     X5E6  ; 2P INFRA WELD REAR#4 CYL' FWD
      OUT     T4241 K1
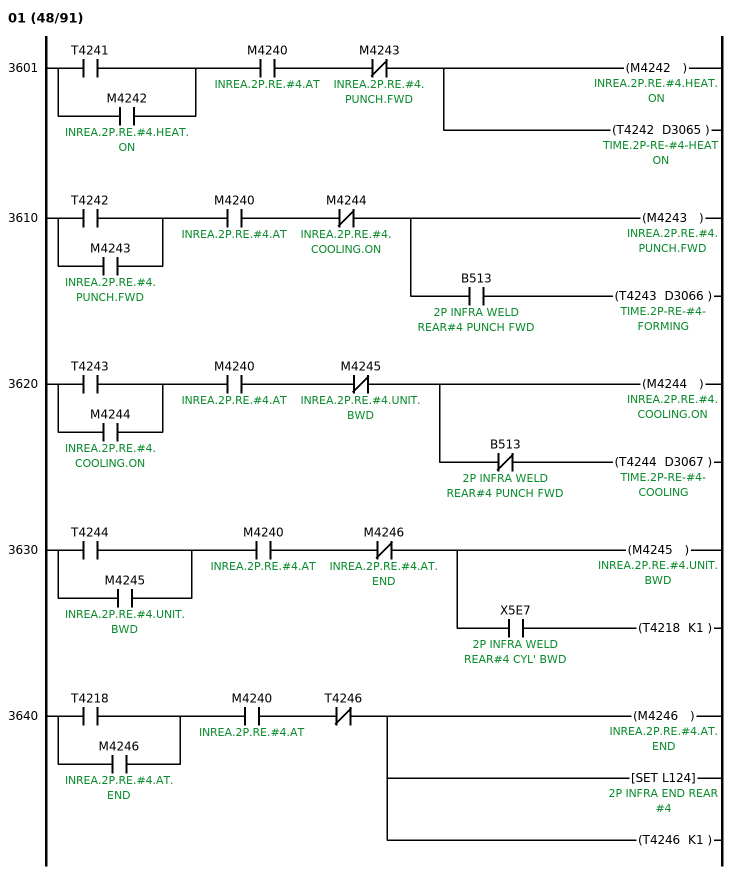
3601  LD      T4241
      OR      M4242  ; INREA.2P.RE.#4.HEAT.ON
      AND     M4240  ; INREA.2P.RE.#4.AT
      ANI     M4243  ; INREA.2P.RE.#4.PUNCH.FWD
      OUT     M4242  ; INREA.2P.RE.#4.HEAT.ON
      OUT     T4242 D3065  ; TIME.2P-RE-#4-HEAT ON
3610  LD      T4242
      OR      M4243  ; INREA.2P.RE.#4.PUNCH.FWD
      AND     M4240  ; INREA.2P.RE.#4.AT
      ANI     M4244  ; INREA.2P.RE.#4.COOLING.ON
      OUT     M4243  ; INREA.2P.RE.#4.PUNCH.FWD
      AND     B513  ; 2P INFRA WELD REAR#4 PUNCH FWD
      OUT     T4243 D3066  ; TIME.2P-RE-#4-FORMING
3620  LD      T4243
      OR      M4244  ; INREA.2P.RE.#4.COOLING.ON
      AND     M4240  ; INREA.2P.RE.#4.AT
      ANI     M4245  ; INREA.2P.RE.#4.UNIT.BWD
      OUT     M4244  ; INREA.2P.RE.#4.COOLING.ON
      ANI     B513  ; 2P INFRA WELD REAR#4 PUNCH FWD
      OUT     T4244 D3067  ; TIME.2P-RE-#4-COOLING
3630  LD      T4244
      OR      M4245  ; INREA.2P.RE.#4.UNIT.BWD
      AND     M4240  ; INREA.2P.RE.#4.AT
      ANI     M4246  ; INREA.2P.RE.#4.AT.END
      OUT     M4245  ; INREA.2P.RE.#4.UNIT.BWD
      AND     X5E7  ; 2P INFRA WELD REAR#4 CYL' BWD
      OUT     T4218 K1
3640  LD      T4218
      OR      M4246  ; INREA.2P.RE.#4.AT.END
      AND     M4240  ; INREA.2P.RE.#4.AT
      ANI     T4246
      OUT     M4246  ; INREA.2P.RE.#4.AT.END
      SET     L124  ; 2P INFRA END REAR #4
      OUT     T4246 K1
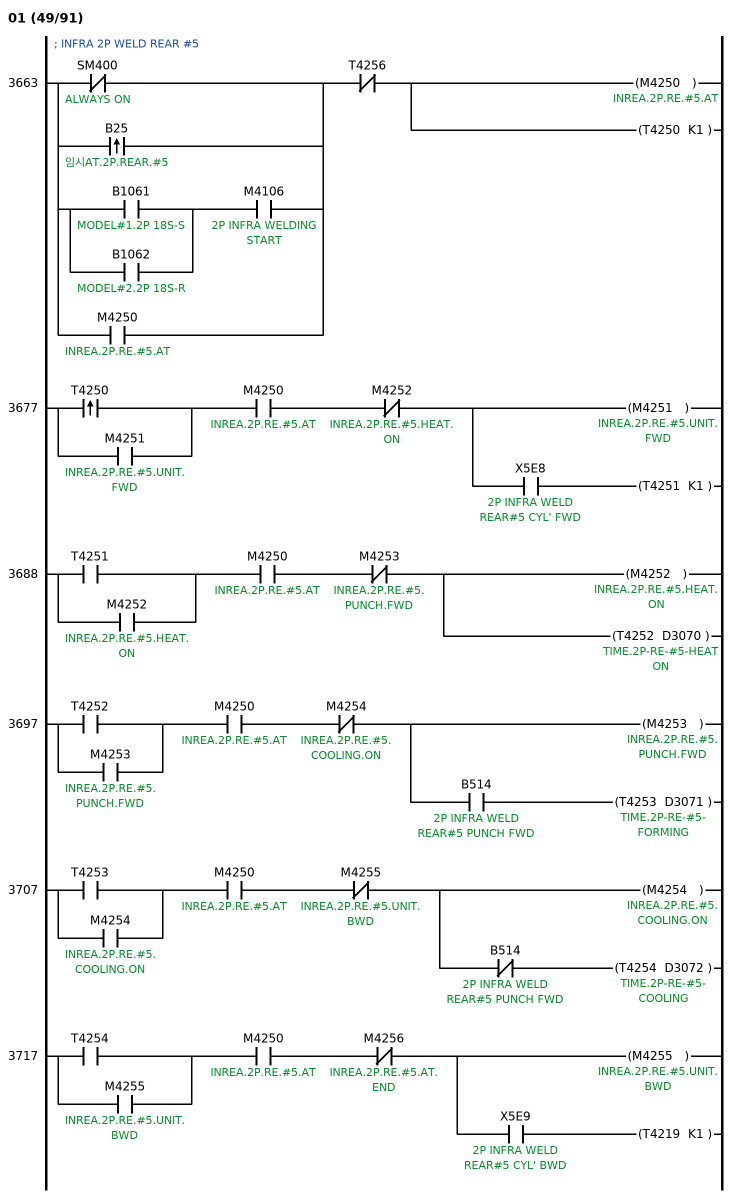
; INFRA 2P WELD REAR #5
3663  LDI     SM400  ; ALWAYS ON
      ORP     B25  ; 임시AT.2P.REAR.#5
      LD      B1061  ; MODEL#1.2P 18S-S
      OR      B1062  ; MODEL#2.2P 18S-R
      AND     M4106  ; 2P INFRA WELDING START
      ORB
      OR      M4250  ; INREA.2P.RE.#5.AT
      ANI     T4256
      OUT     M4250  ; INREA.2P.RE.#5.AT
      OUT     T4250 K1
3677  LDP     T4250
      OR      M4251  ; INREA.2P.RE.#5.UNIT.FWD
      AND     M4250  ; INREA.2P.RE.#5.AT
      ANI     M4252  ; INREA.2P.RE.#5.HEAT.ON
      OUT     M4251  ; INREA.2P.RE.#5.UNIT.FWD
      AND     X5E8  ; 2P INFRA WELD REAR#5 CYL' FWD
      OUT     T4251 K1
3688  LD      T4251
      OR      M4252  ; INREA.2P.RE.#5.HEAT.ON
      AND     M4250  ; INREA.2P.RE.#5.AT
      ANI     M4253  ; INREA.2P.RE.#5.PUNCH.FWD
      OUT     M4252  ; INREA.2P.RE.#5.HEAT.ON
      OUT     T4252 D3070  ; TIME.2P-RE-#5-HEAT ON
3697  LD      T4252
      OR      M4253  ; INREA.2P.RE.#5.PUNCH.FWD
      AND     M4250  ; INREA.2P.RE.#5.AT
      ANI     M4254  ; INREA.2P.RE.#5.COOLING.ON
      OUT     M4253  ; INREA.2P.RE.#5.PUNCH.FWD
      AND     B514  ; 2P INFRA WELD REAR#5 PUNCH FWD
      OUT     T4253 D3071  ; TIME.2P-RE-#5-FORMING
3707  LD      T4253
      OR      M4254  ; INREA.2P.RE.#5.COOLING.ON
      AND     M4250  ; INREA.2P.RE.#5.AT
      ANI     M4255  ; INREA.2P.RE.#5.UNIT.BWD
      OUT     M4254  ; INREA.2P.RE.#5.COOLING.ON
      ANI     B514  ; 2P INFRA WELD REAR#5 PUNCH FWD
      OUT     T4254 D3072  ; TIME.2P-RE-#5-COOLING
3717  LD      T4254
      OR      M4255  ; INREA.2P.RE.#5.UNIT.BWD
      AND     M4250  ; INREA.2P.RE.#5.AT
      ANI     M4256  ; INREA.2P.RE.#5.AT.END
      OUT     M4255  ; INREA.2P.RE.#5.UNIT.BWD
      AND     X5E9  ; 2P INFRA WELD REAR#5 CYL' BWD
      OUT     T4219 K1
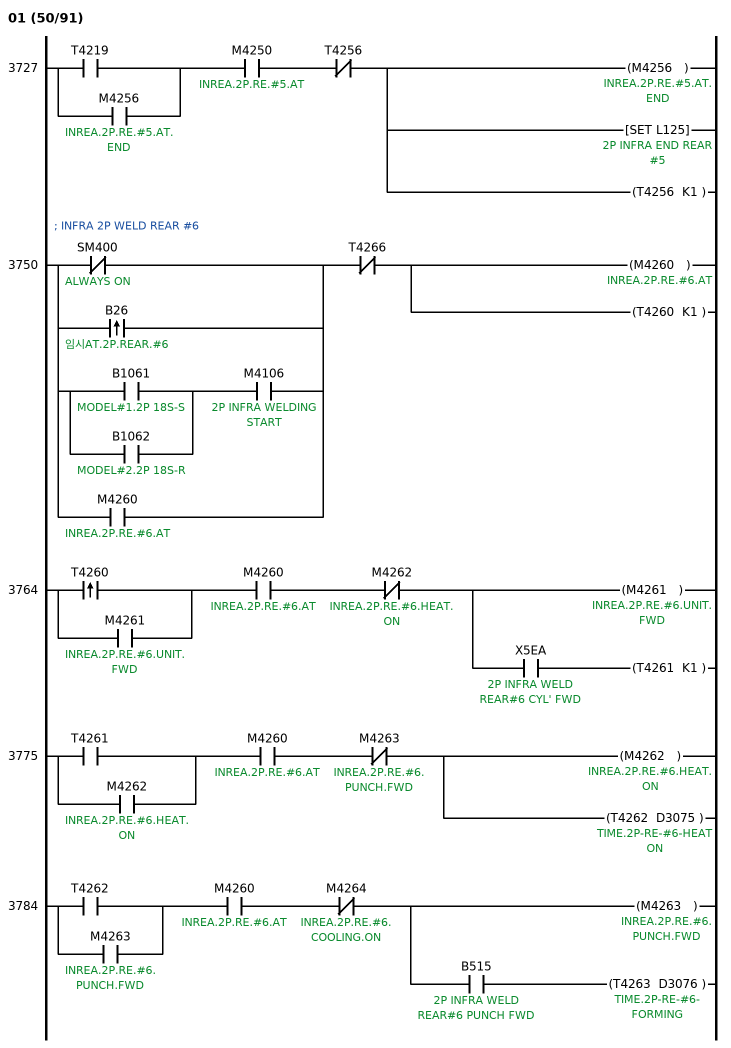
3727  LD      T4219
      OR      M4256  ; INREA.2P.RE.#5.AT.END
      AND     M4250  ; INREA.2P.RE.#5.AT
      ANI     T4256
      OUT     M4256  ; INREA.2P.RE.#5.AT.END
      SET     L125  ; 2P INFRA END REAR #5
      OUT     T4256 K1
; INFRA 2P WELD REAR #6
3750  LDI     SM400  ; ALWAYS ON
      ORP     B26  ; 임시AT.2P.REAR.#6
      LD      B1061  ; MODEL#1.2P 18S-S
      OR      B1062  ; MODEL#2.2P 18S-R
      AND     M4106  ; 2P INFRA WELDING START
      ORB
      OR      M4260  ; INREA.2P.RE.#6.AT
      ANI     T4266
      OUT     M4260  ; INREA.2P.RE.#6.AT
      OUT     T4260 K1
3764  LDP     T4260
      OR      M4261  ; INREA.2P.RE.#6.UNIT.FWD
      AND     M4260  ; INREA.2P.RE.#6.AT
      ANI     M4262  ; INREA.2P.RE.#6.HEAT.ON
      OUT     M4261  ; INREA.2P.RE.#6.UNIT.FWD
      AND     X5EA  ; 2P INFRA WELD REAR#6 CYL' FWD
      OUT     T4261 K1
3775  LD      T4261
      OR      M4262  ; INREA.2P.RE.#6.HEAT.ON
      AND     M4260  ; INREA.2P.RE.#6.AT
      ANI     M4263  ; INREA.2P.RE.#6.PUNCH.FWD
      OUT     M4262  ; INREA.2P.RE.#6.HEAT.ON
      OUT     T4262 D3075  ; TIME.2P-RE-#6-HEAT ON
3784  LD      T4262
      OR      M4263  ; INREA.2P.RE.#6.PUNCH.FWD
      AND     M4260  ; INREA.2P.RE.#6.AT
      ANI     M4264  ; INREA.2P.RE.#6.COOLING.ON
      OUT     M4263  ; INREA.2P.RE.#6.PUNCH.FWD
      AND     B515  ; 2P INFRA WELD REAR#6 PUNCH FWD
      OUT     T4263 D3076  ; TIME.2P-RE-#6-FORMING
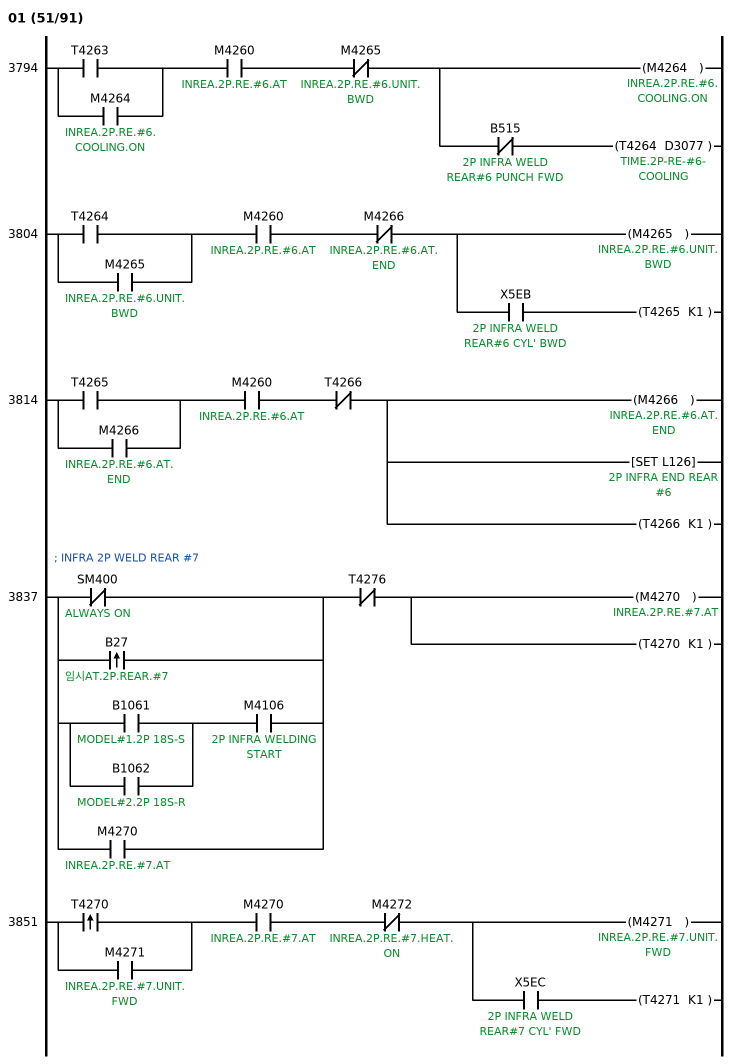
3794  LD      T4263
      OR      M4264  ; INREA.2P.RE.#6.COOLING.ON
      AND     M4260  ; INREA.2P.RE.#6.AT
      ANI     M4265  ; INREA.2P.RE.#6.UNIT.BWD
      OUT     M4264  ; INREA.2P.RE.#6.COOLING.ON
      ANI     B515  ; 2P INFRA WELD REAR#6 PUNCH FWD
      OUT     T4264 D3077  ; TIME.2P-RE-#6-COOLING
3804  LD      T4264
      OR      M4265  ; INREA.2P.RE.#6.UNIT.BWD
      AND     M4260  ; INREA.2P.RE.#6.AT
      ANI     M4266  ; INREA.2P.RE.#6.AT.END
      OUT     M4265  ; INREA.2P.RE.#6.UNIT.BWD
      AND     X5EB  ; 2P INFRA WELD REAR#6 CYL' BWD
      OUT     T4265 K1
3814  LD      T4265
      OR      M4266  ; INREA.2P.RE.#6.AT.END
      AND     M4260  ; INREA.2P.RE.#6.AT
      ANI     T4266
      OUT     M4266  ; INREA.2P.RE.#6.AT.END
      SET     L126  ; 2P INFRA END REAR #6
      OUT     T4266 K1
; INFRA 2P WELD REAR #7
3837  LDI     SM400  ; ALWAYS ON
      ORP     B27  ; 임시AT.2P.REAR.#7
      LD      B1061  ; MODEL#1.2P 18S-S
      OR      B1062  ; MODEL#2.2P 18S-R
      AND     M4106  ; 2P INFRA WELDING START
      ORB
      OR      M4270  ; INREA.2P.RE.#7.AT
      ANI     T4276
      OUT     M4270  ; INREA.2P.RE.#7.AT
      OUT     T4270 K1
3851  LDP     T4270
      OR      M4271  ; INREA.2P.RE.#7.UNIT.FWD
      AND     M4270  ; INREA.2P.RE.#7.AT
      ANI     M4272  ; INREA.2P.RE.#7.HEAT.ON
      OUT     M4271  ; INREA.2P.RE.#7.UNIT.FWD
      AND     X5EC  ; 2P INFRA WELD REAR#7 CYL' FWD
      OUT     T4271 K1
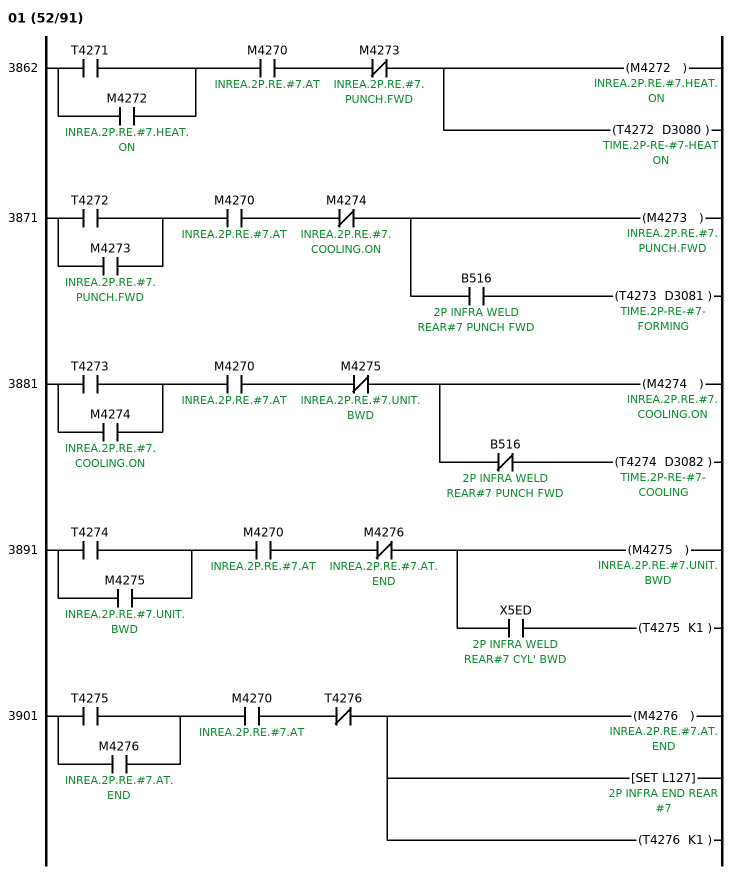
3862  LD      T4271
      OR      M4272  ; INREA.2P.RE.#7.HEAT.ON
      AND     M4270  ; INREA.2P.RE.#7.AT
      ANI     M4273  ; INREA.2P.RE.#7.PUNCH.FWD
      OUT     M4272  ; INREA.2P.RE.#7.HEAT.ON
      OUT     T4272 D3080  ; TIME.2P-RE-#7-HEAT ON
3871  LD      T4272
      OR      M4273  ; INREA.2P.RE.#7.PUNCH.FWD
      AND     M4270  ; INREA.2P.RE.#7.AT
      ANI     M4274  ; INREA.2P.RE.#7.COOLING.ON
      OUT     M4273  ; INREA.2P.RE.#7.PUNCH.FWD
      AND     B516  ; 2P INFRA WELD REAR#7 PUNCH FWD
      OUT     T4273 D3081  ; TIME.2P-RE-#7-FORMING
3881  LD      T4273
      OR      M4274  ; INREA.2P.RE.#7.COOLING.ON
      AND     M4270  ; INREA.2P.RE.#7.AT
      ANI     M4275  ; INREA.2P.RE.#7.UNIT.BWD
      OUT     M4274  ; INREA.2P.RE.#7.COOLING.ON
      ANI     B516  ; 2P INFRA WELD REAR#7 PUNCH FWD
      OUT     T4274 D3082  ; TIME.2P-RE-#7-COOLING
3891  LD      T4274
      OR      M4275  ; INREA.2P.RE.#7.UNIT.BWD
      AND     M4270  ; INREA.2P.RE.#7.AT
      ANI     M4276  ; INREA.2P.RE.#7.AT.END
      OUT     M4275  ; INREA.2P.RE.#7.UNIT.BWD
      AND     X5ED  ; 2P INFRA WELD REAR#7 CYL' BWD
      OUT     T4275 K1
3901  LD      T4275
      OR      M4276  ; INREA.2P.RE.#7.AT.END
      AND     M4270  ; INREA.2P.RE.#7.AT
      ANI     T4276
      OUT     M4276  ; INREA.2P.RE.#7.AT.END
      SET     L127  ; 2P INFRA END REAR #7
      OUT     T4276 K1
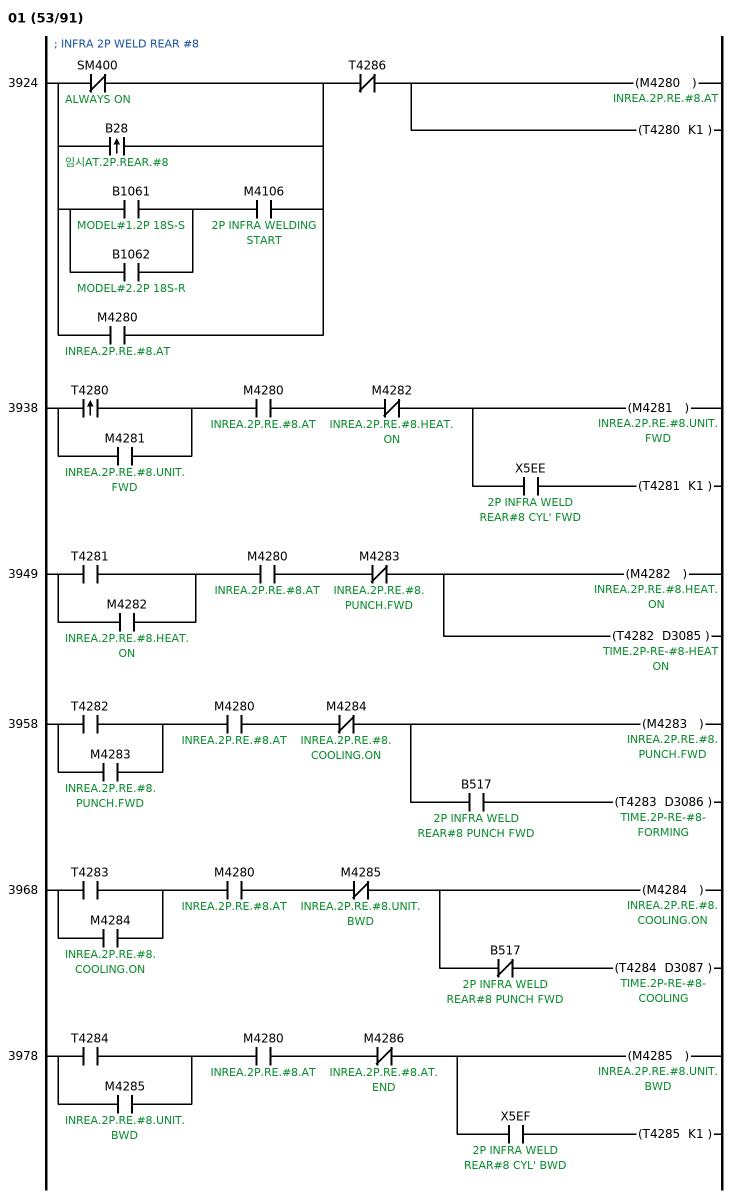
; INFRA 2P WELD REAR #8
3924  LDI     SM400  ; ALWAYS ON
      ORP     B28  ; 임시AT.2P.REAR.#8
      LD      B1061  ; MODEL#1.2P 18S-S
      OR      B1062  ; MODEL#2.2P 18S-R
      AND     M4106  ; 2P INFRA WELDING START
      ORB
      OR      M4280  ; INREA.2P.RE.#8.AT
      ANI     T4286
      OUT     M4280  ; INREA.2P.RE.#8.AT
      OUT     T4280 K1
3938  LDP     T4280
      OR      M4281  ; INREA.2P.RE.#8.UNIT.FWD
      AND     M4280  ; INREA.2P.RE.#8.AT
      ANI     M4282  ; INREA.2P.RE.#8.HEAT.ON
      OUT     M4281  ; INREA.2P.RE.#8.UNIT.FWD
      AND     X5EE  ; 2P INFRA WELD REAR#8 CYL' FWD
      OUT     T4281 K1
3949  LD      T4281
      OR      M4282  ; INREA.2P.RE.#8.HEAT.ON
      AND     M4280  ; INREA.2P.RE.#8.AT
      ANI     M4283  ; INREA.2P.RE.#8.PUNCH.FWD
      OUT     M4282  ; INREA.2P.RE.#8.HEAT.ON
      OUT     T4282 D3085  ; TIME.2P-RE-#8-HEAT ON
3958  LD      T4282
      OR      M4283  ; INREA.2P.RE.#8.PUNCH.FWD
      AND     M4280  ; INREA.2P.RE.#8.AT
      ANI     M4284  ; INREA.2P.RE.#8.COOLING.ON
      OUT     M4283  ; INREA.2P.RE.#8.PUNCH.FWD
      AND     B517  ; 2P INFRA WELD REAR#8 PUNCH FWD
      OUT     T4283 D3086  ; TIME.2P-RE-#8-FORMING
3968  LD      T4283
      OR      M4284  ; INREA.2P.RE.#8.COOLING.ON
      AND     M4280  ; INREA.2P.RE.#8.AT
      ANI     M4285  ; INREA.2P.RE.#8.UNIT.BWD
      OUT     M4284  ; INREA.2P.RE.#8.COOLING.ON
      ANI     B517  ; 2P INFRA WELD REAR#8 PUNCH FWD
      OUT     T4284 D3087  ; TIME.2P-RE-#8-COOLING
3978  LD      T4284
      OR      M4285  ; INREA.2P.RE.#8.UNIT.BWD
      AND     M4280  ; INREA.2P.RE.#8.AT
      ANI     M4286  ; INREA.2P.RE.#8.AT.END
      OUT     M4285  ; INREA.2P.RE.#8.UNIT.BWD
      AND     X5EF  ; 2P INFRA WELD REAR#8 CYL' BWD
      OUT     T4285 K1
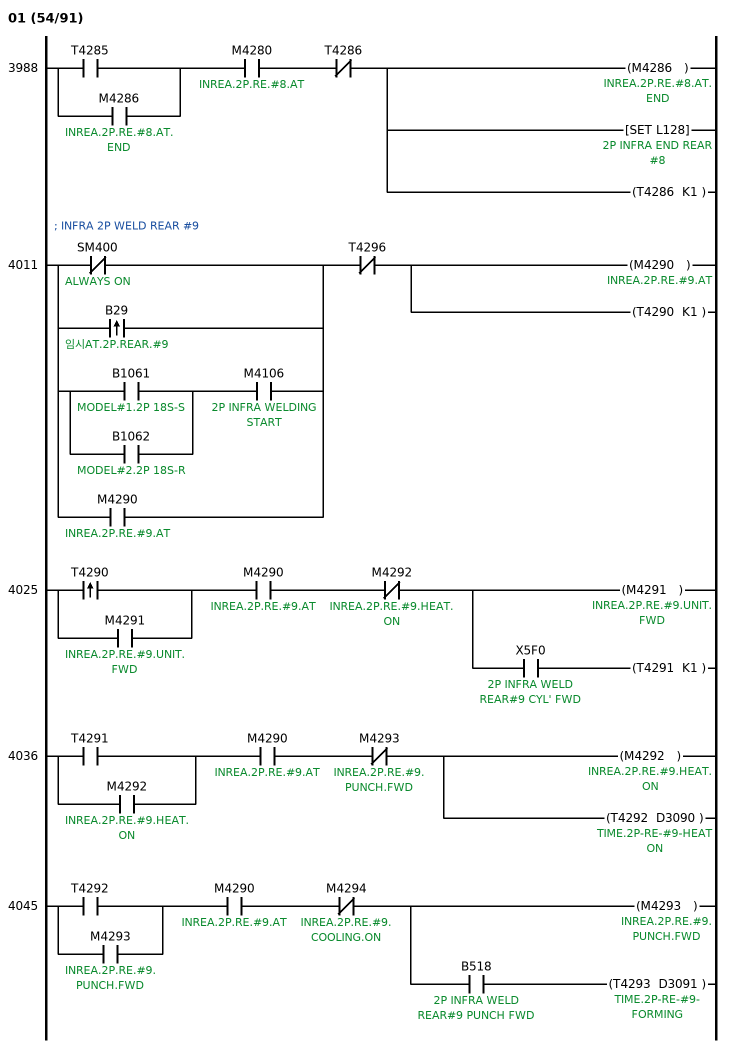
3988  LD      T4285
      OR      M4286  ; INREA.2P.RE.#8.AT.END
      AND     M4280  ; INREA.2P.RE.#8.AT
      ANI     T4286
      OUT     M4286  ; INREA.2P.RE.#8.AT.END
      SET     L128  ; 2P INFRA END REAR #8
      OUT     T4286 K1
; INFRA 2P WELD REAR #9
4011  LDI     SM400  ; ALWAYS ON
      ORP     B29  ; 임시AT.2P.REAR.#9
      LD      B1061  ; MODEL#1.2P 18S-S
      OR      B1062  ; MODEL#2.2P 18S-R
      AND     M4106  ; 2P INFRA WELDING START
      ORB
      OR      M4290  ; INREA.2P.RE.#9.AT
      ANI     T4296
      OUT     M4290  ; INREA.2P.RE.#9.AT
      OUT     T4290 K1
4025  LDP     T4290
      OR      M4291  ; INREA.2P.RE.#9.UNIT.FWD
      AND     M4290  ; INREA.2P.RE.#9.AT
      ANI     M4292  ; INREA.2P.RE.#9.HEAT.ON
      OUT     M4291  ; INREA.2P.RE.#9.UNIT.FWD
      AND     X5F0  ; 2P INFRA WELD REAR#9 CYL' FWD
      OUT     T4291 K1
4036  LD      T4291
      OR      M4292  ; INREA.2P.RE.#9.HEAT.ON
      AND     M4290  ; INREA.2P.RE.#9.AT
      ANI     M4293  ; INREA.2P.RE.#9.PUNCH.FWD
      OUT     M4292  ; INREA.2P.RE.#9.HEAT.ON
      OUT     T4292 D3090  ; TIME.2P-RE-#9-HEAT ON
4045  LD      T4292
      OR      M4293  ; INREA.2P.RE.#9.PUNCH.FWD
      AND     M4290  ; INREA.2P.RE.#9.AT
      ANI     M4294  ; INREA.2P.RE.#9.COOLING.ON
      OUT     M4293  ; INREA.2P.RE.#9.PUNCH.FWD
      AND     B518  ; 2P INFRA WELD REAR#9 PUNCH FWD
      OUT     T4293 D3091  ; TIME.2P-RE-#9-FORMING
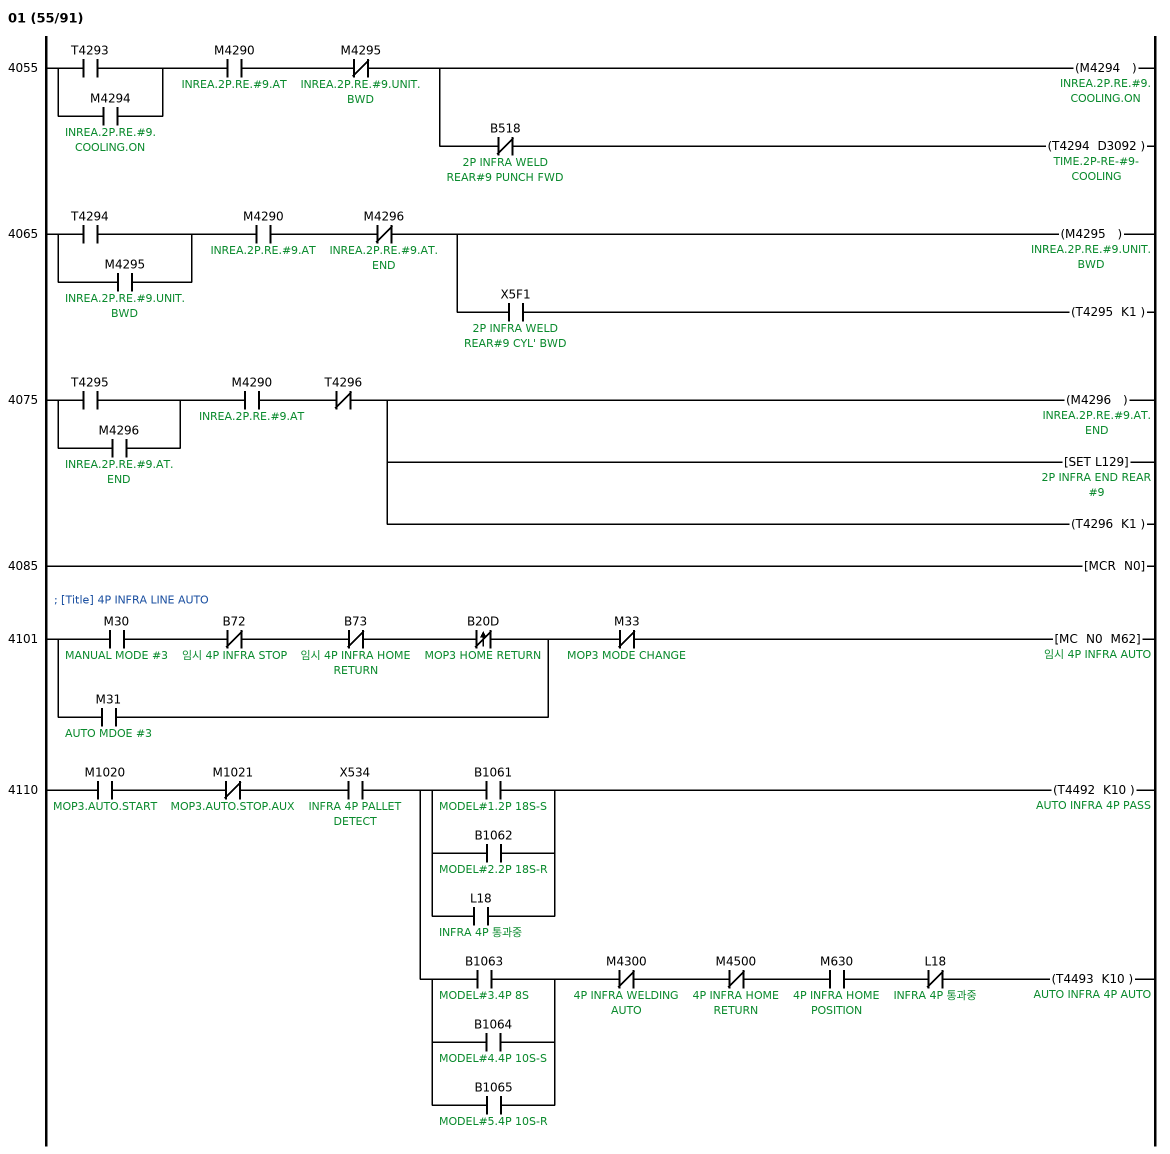
4055  LD      T4293
      OR      M4294  ; INREA.2P.RE.#9.COOLING.ON
      AND     M4290  ; INREA.2P.RE.#9.AT
      ANI     M4295  ; INREA.2P.RE.#9.UNIT.BWD
      OUT     M4294  ; INREA.2P.RE.#9.COOLING.ON
      ANI     B518  ; 2P INFRA WELD REAR#9 PUNCH FWD
      OUT     T4294 D3092  ; TIME.2P-RE-#9-COOLING
4065  LD      T4294
      OR      M4295  ; INREA.2P.RE.#9.UNIT.BWD
      AND     M4290  ; INREA.2P.RE.#9.AT
      ANI     M4296  ; INREA.2P.RE.#9.AT.END
      OUT     M4295  ; INREA.2P.RE.#9.UNIT.BWD
      AND     X5F1  ; 2P INFRA WELD REAR#9 CYL' BWD
      OUT     T4295 K1
4075  LD      T4295
      OR      M4296  ; INREA.2P.RE.#9.AT.END
      AND     M4290  ; INREA.2P.RE.#9.AT
      ANI     T4296
      OUT     M4296  ; INREA.2P.RE.#9.AT.END
      SET     L129  ; 2P INFRA END REAR #9
      OUT     T4296 K1
4085  MCR     N0
; [Title] 4P INFRA LINE AUTO
4101  LD      M30  ; MANUAL MODE #3
      ANI     B72  ; 임시 4P INFRA STOP
      ANI     B73  ; 임시 4P INFRA HOME RETURN
      ANDPI   B20D  ; MOP3 HOME RETURN
      OR      M31  ; AUTO MDOE #3
      ANI     M33  ; MOP3 MODE CHANGE
      MC      N0 M62  ; 임시 4P INFRA AUTO
4110  LD      M1020  ; MOP3.AUTO.START
      ANI     M1021  ; MOP3.AUTO.STOP.AUX
      AND     X534  ; INFRA 4P PALLET DETECT
      MPS
      LD      B1061  ; MODEL#1.2P 18S-S
      OR      B1062  ; MODEL#2.2P 18S-R
      OR      L18  ; INFRA 4P 통과중
      ANB
      OUT     T4492 K10  ; AUTO INFRA 4P PASS
      MPP
      LD      B1063  ; MODEL#3.4P 8S
      OR      B1064  ; MODEL#4.4P 10S-S
      OR      B1065  ; MODEL#5.4P 10S-R
      ANB
      ANI     M4300  ; 4P INFRA WELDING AUTO
      ANI     M4500  ; 4P INFRA HOME RETURN
      AND     M630  ; 4P INFRA HOME POSITION
      ANI     L18  ; INFRA 4P 통과중
      OUT     T4493 K10  ; AUTO INFRA 4P AUTO
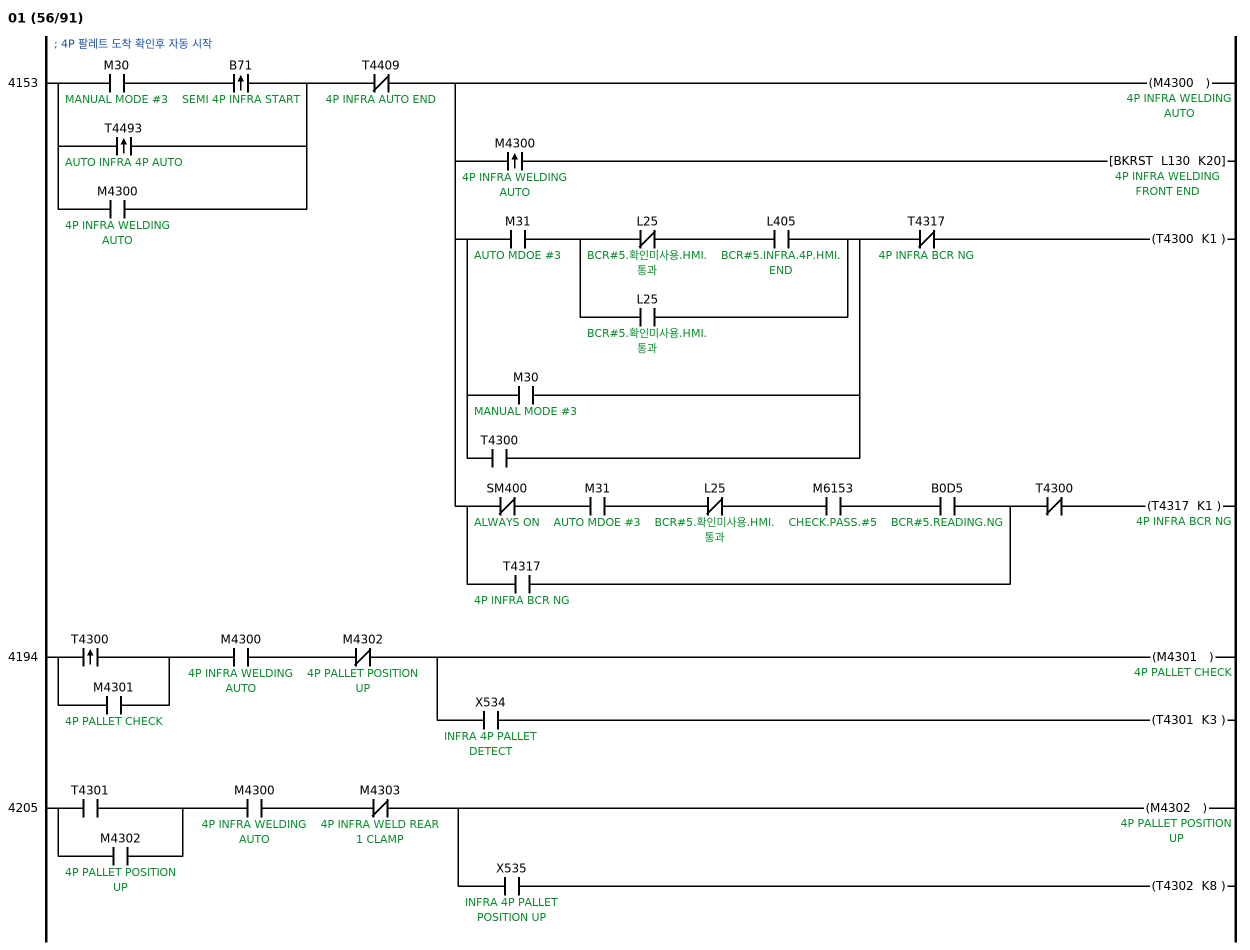
; 4P 팔레트 도착 확인후 자동 시작
4153  LD      M30  ; MANUAL MODE #3
      ANDP    B71  ; SEMI 4P INFRA START
      ORP     T4493  ; AUTO INFRA 4P AUTO
      OR      M4300  ; 4P INFRA WELDING AUTO
      ANI     T4409  ; 4P INFRA AUTO END
      OUT     M4300  ; 4P INFRA WELDING AUTO
      MPS
      ANDP    M4300  ; 4P INFRA WELDING AUTO
      BKRST   L130 K20  ; 4P INFRA WELDING FRONT END
      MRD
      LD      M31  ; AUTO MDOE #3
      LDI     L25  ; BCR#5.확인미사용.HMI.통과
      AND     L405  ; BCR#5.INFRA.4P.HMI.END
      OR      L25  ; BCR#5.확인미사용.HMI.통과
      ANB
      OR      M30  ; MANUAL MODE #3
      OR      T4300
      ANB
      ANI     T4317  ; 4P INFRA BCR NG
      OUT     T4300 K1
      MPP
      LDI     SM400  ; ALWAYS ON
      AND     M31  ; AUTO MDOE #3
      ANI     L25  ; BCR#5.확인미사용.HMI.통과
      AND     M6153  ; CHECK.PASS.#5
      AND     B0D5  ; BCR#5.READING.NG
      OR      T4317  ; 4P INFRA BCR NG
      ANB
      ANI     T4300
      OUT     T4317 K1  ; 4P INFRA BCR NG
4194  LDP     T4300
      OR      M4301  ; 4P PALLET CHECK
      AND     M4300  ; 4P INFRA WELDING AUTO
      ANI     M4302  ; 4P PALLET POSITION UP
      OUT     M4301  ; 4P PALLET CHECK
      AND     X534  ; INFRA 4P PALLET DETECT
      OUT     T4301 K3
4205  LD      T4301
      OR      M4302  ; 4P PALLET POSITION UP
      AND     M4300  ; 4P INFRA WELDING AUTO
      ANI     M4303  ; 4P INFRA WELD REAR 1 CLAMP
      OUT     M4302  ; 4P PALLET POSITION UP
      AND     X535  ; INFRA 4P PALLET POSITION UP
      OUT     T4302 K8
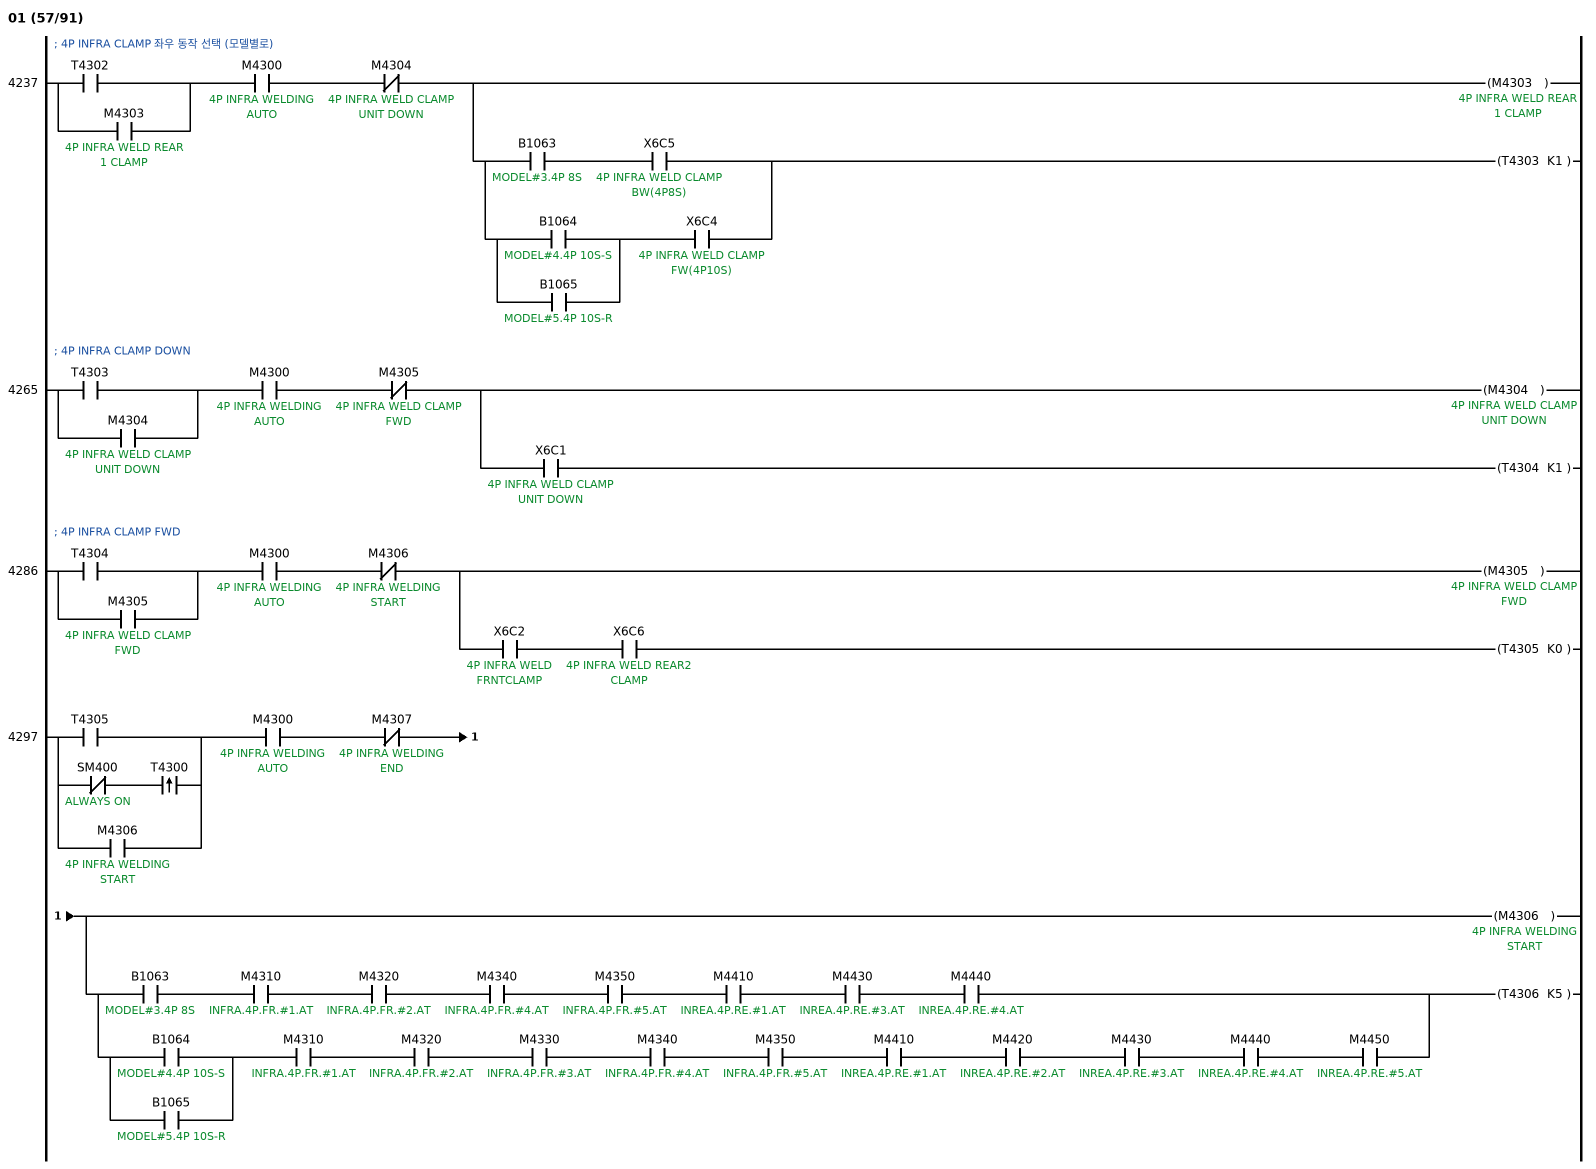
; 4P INFRA CLAMP 좌우 동작 선택 (모델별로)
4237  LD      T4302
      OR      M4303  ; 4P INFRA WELD REAR 1 CLAMP
      AND     M4300  ; 4P INFRA WELDING AUTO
      ANI     M4304  ; 4P INFRA WELD CLAMP UNIT DOWN
      OUT     M4303  ; 4P INFRA WELD REAR 1 CLAMP
      LD      B1063  ; MODEL#3.4P 8S
      AND     X6C5  ; 4P INFRA WELD CLAMP BW(4P8S)
      LD      B1064  ; MODEL#4.4P 10S-S
      OR      B1065  ; MODEL#5.4P 10S-R
      AND     X6C4  ; 4P INFRA WELD CLAMP FW(4P10S)
      ORB
      ANB
      OUT     T4303 K1
; 4P INFRA CLAMP DOWN
4265  LD      T4303
      OR      M4304  ; 4P INFRA WELD CLAMP UNIT DOWN
      AND     M4300  ; 4P INFRA WELDING AUTO
      ANI     M4305  ; 4P INFRA WELD CLAMP FWD
      OUT     M4304  ; 4P INFRA WELD CLAMP UNIT DOWN
      AND     X6C1  ; 4P INFRA WELD CLAMP UNIT DOWN
      OUT     T4304 K1
; 4P INFRA CLAMP FWD
4286  LD      T4304
      OR      M4305  ; 4P INFRA WELD CLAMP FWD
      AND     M4300  ; 4P INFRA WELDING AUTO
      ANI     M4306  ; 4P INFRA WELDING START
      OUT     M4305  ; 4P INFRA WELD CLAMP FWD
      AND     X6C2  ; 4P INFRA WELD FRNTCLAMP
      AND     X6C6  ; 4P INFRA WELD REAR2 CLAMP
      OUT     T4305 K0
4297  LD      T4305
      LDI     SM400  ; ALWAYS ON
      ANDP    T4300
      ORB
      OR      M4306  ; 4P INFRA WELDING START
      AND     M4300  ; 4P INFRA WELDING AUTO
      ANI     M4307  ; 4P INFRA WELDING END
      OUT     M4306  ; 4P INFRA WELDING START
      LD      B1063  ; MODEL#3.4P 8S
      AND     M4310  ; INFRA.4P.FR.#1.AT
      AND     M4320  ; INFRA.4P.FR.#2.AT
      AND     M4340  ; INFRA.4P.FR.#4.AT
      AND     M4350  ; INFRA.4P.FR.#5.AT
      AND     M4410  ; INREA.4P.RE.#1.AT
      AND     M4430  ; INREA.4P.RE.#3.AT
      AND     M4440  ; INREA.4P.RE.#4.AT
      LD      B1064  ; MODEL#4.4P 10S-S
      OR      B1065  ; MODEL#5.4P 10S-R
      AND     M4310  ; INFRA.4P.FR.#1.AT
      AND     M4320  ; INFRA.4P.FR.#2.AT
      AND     M4330  ; INFRA.4P.FR.#3.AT
      AND     M4340  ; INFRA.4P.FR.#4.AT
      AND     M4350  ; INFRA.4P.FR.#5.AT
      AND     M4410  ; INREA.4P.RE.#1.AT
      AND     M4420  ; INREA.4P.RE.#2.AT
      AND     M4430  ; INREA.4P.RE.#3.AT
      AND     M4440  ; INREA.4P.RE.#4.AT
      AND     M4450  ; INREA.4P.RE.#5.AT
      ORB
      ANB
      OUT     T4306 K5
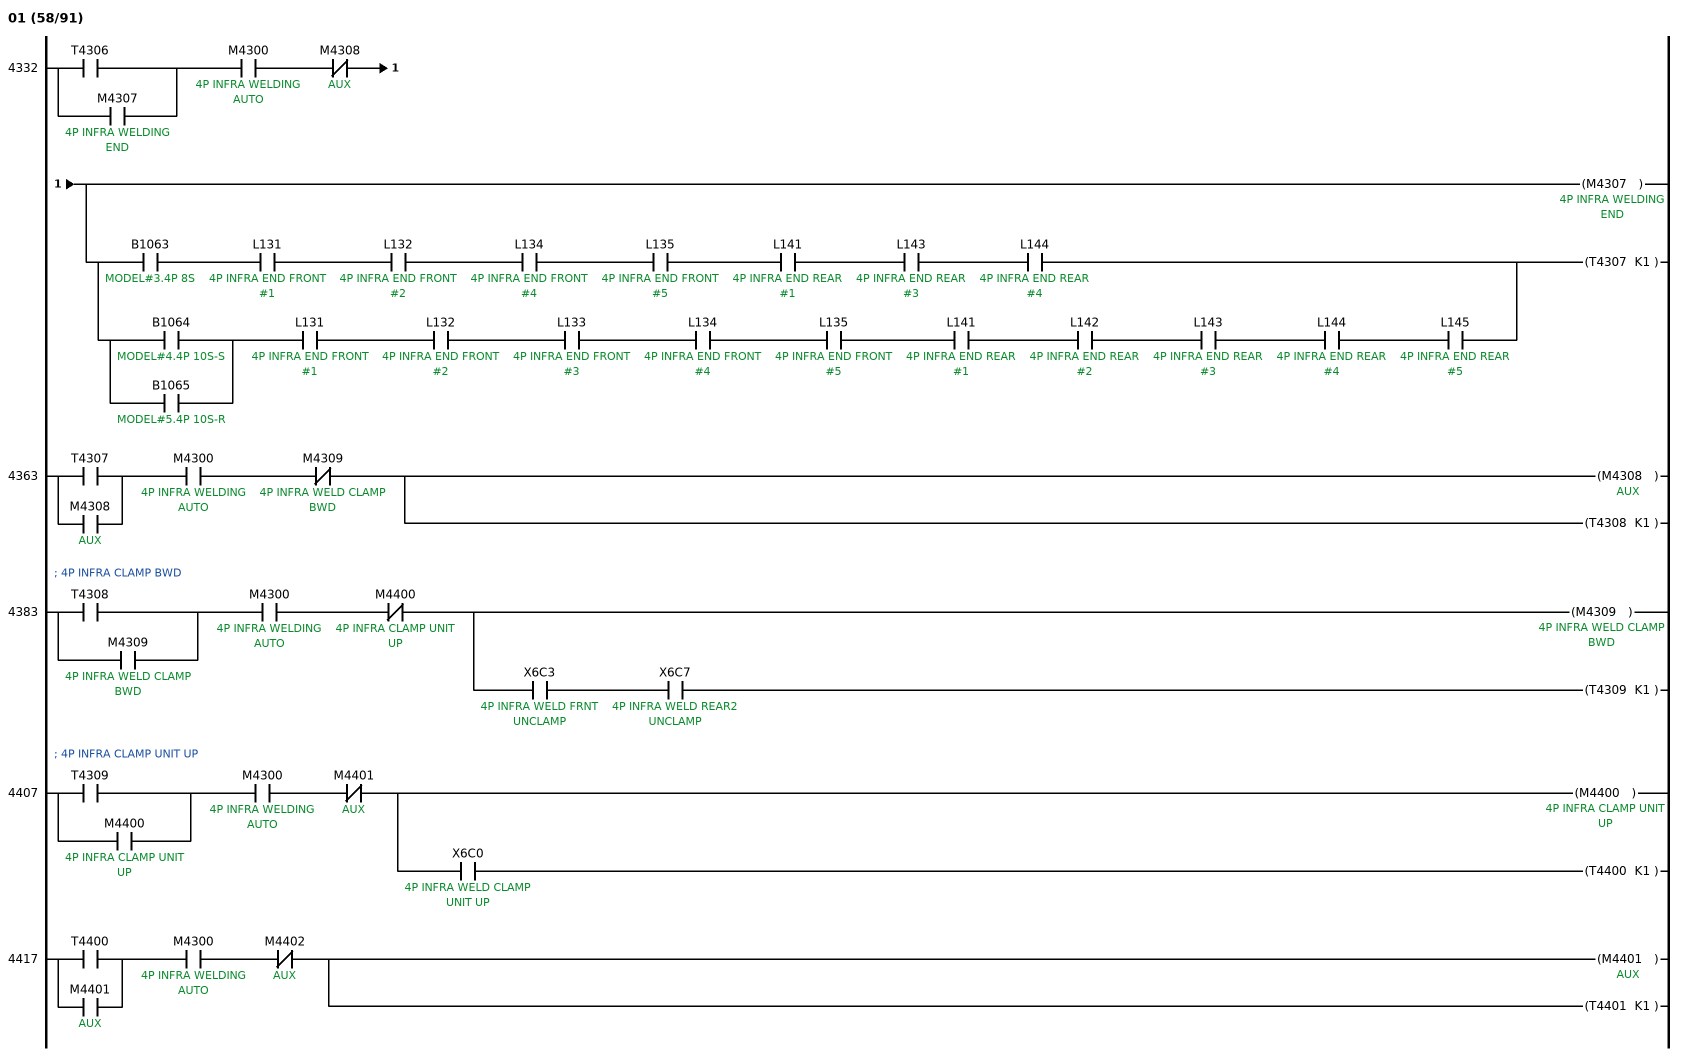
4332  LD      T4306
      OR      M4307  ; 4P INFRA WELDING END
      AND     M4300  ; 4P INFRA WELDING AUTO
      ANI     M4308  ; AUX
      OUT     M4307  ; 4P INFRA WELDING END
      LD      B1063  ; MODEL#3.4P 8S
      AND     L131  ; 4P INFRA END FRONT #1
      AND     L132  ; 4P INFRA END FRONT #2
      AND     L134  ; 4P INFRA END FRONT #4
      AND     L135  ; 4P INFRA END FRONT #5
      AND     L141  ; 4P INFRA END REAR #1
      AND     L143  ; 4P INFRA END REAR #3
      AND     L144  ; 4P INFRA END REAR #4
      LD      B1064  ; MODEL#4.4P 10S-S
      OR      B1065  ; MODEL#5.4P 10S-R
      AND     L131  ; 4P INFRA END FRONT #1
      AND     L132  ; 4P INFRA END FRONT #2
      AND     L133  ; 4P INFRA END FRONT #3
      AND     L134  ; 4P INFRA END FRONT #4
      AND     L135  ; 4P INFRA END FRONT #5
      AND     L141  ; 4P INFRA END REAR #1
      AND     L142  ; 4P INFRA END REAR #2
      AND     L143  ; 4P INFRA END REAR #3
      AND     L144  ; 4P INFRA END REAR #4
      AND     L145  ; 4P INFRA END REAR #5
      ORB
      ANB
      OUT     T4307 K1
4363  LD      T4307
      OR      M4308  ; AUX
      AND     M4300  ; 4P INFRA WELDING AUTO
      ANI     M4309  ; 4P INFRA WELD CLAMP BWD
      OUT     M4308  ; AUX
      OUT     T4308 K1
; 4P INFRA CLAMP BWD
4383  LD      T4308
      OR      M4309  ; 4P INFRA WELD CLAMP BWD
      AND     M4300  ; 4P INFRA WELDING AUTO
      ANI     M4400  ; 4P INFRA CLAMP UNIT UP
      OUT     M4309  ; 4P INFRA WELD CLAMP BWD
      AND     X6C3  ; 4P INFRA WELD FRNT UNCLAMP
      AND     X6C7  ; 4P INFRA WELD REAR2 UNCLAMP
      OUT     T4309 K1
; 4P INFRA CLAMP UNIT UP
4407  LD      T4309
      OR      M4400  ; 4P INFRA CLAMP UNIT UP
      AND     M4300  ; 4P INFRA WELDING AUTO
      ANI     M4401  ; AUX
      OUT     M4400  ; 4P INFRA CLAMP UNIT UP
      AND     X6C0  ; 4P INFRA WELD CLAMP UNIT UP
      OUT     T4400 K1
4417  LD      T4400
      OR      M4401  ; AUX
      AND     M4300  ; 4P INFRA WELDING AUTO
      ANI     M4402  ; AUX
      OUT     M4401  ; AUX
      OUT     T4401 K1
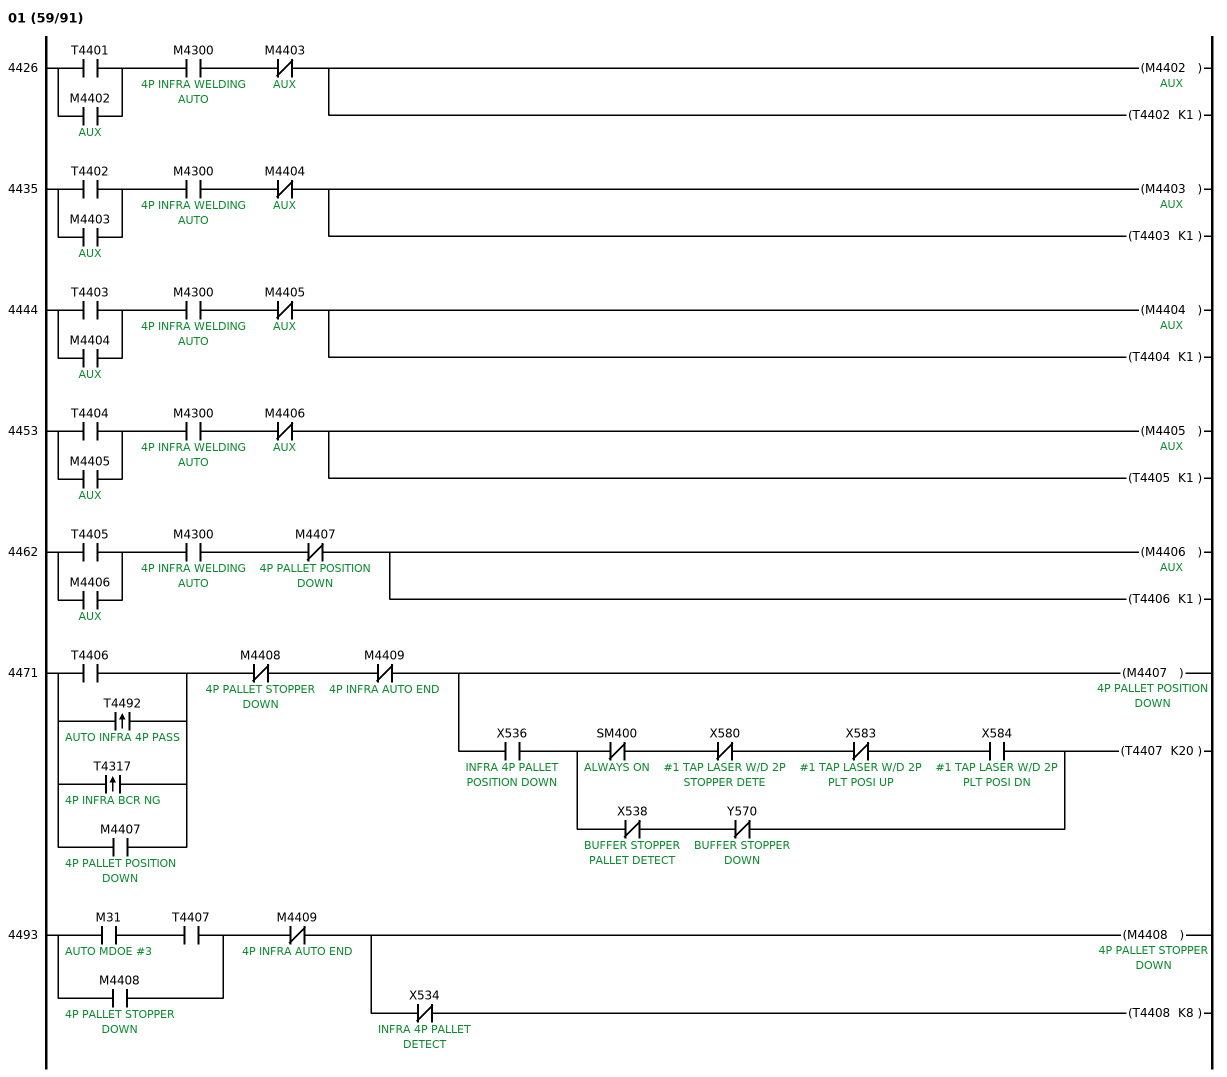
4426  LD      T4401
      OR      M4402  ; AUX
      AND     M4300  ; 4P INFRA WELDING AUTO
      ANI     M4403  ; AUX
      OUT     M4402  ; AUX
      OUT     T4402 K1
4435  LD      T4402
      OR      M4403  ; AUX
      AND     M4300  ; 4P INFRA WELDING AUTO
      ANI     M4404  ; AUX
      OUT     M4403  ; AUX
      OUT     T4403 K1
4444  LD      T4403
      OR      M4404  ; AUX
      AND     M4300  ; 4P INFRA WELDING AUTO
      ANI     M4405  ; AUX
      OUT     M4404  ; AUX
      OUT     T4404 K1
4453  LD      T4404
      OR      M4405  ; AUX
      AND     M4300  ; 4P INFRA WELDING AUTO
      ANI     M4406  ; AUX
      OUT     M4405  ; AUX
      OUT     T4405 K1
4462  LD      T4405
      OR      M4406  ; AUX
      AND     M4300  ; 4P INFRA WELDING AUTO
      ANI     M4407  ; 4P PALLET POSITION DOWN
      OUT     M4406  ; AUX
      OUT     T4406 K1
4471  LD      T4406
      ORP     T4492  ; AUTO INFRA 4P PASS
      ORP     T4317  ; 4P INFRA BCR NG
      OR      M4407  ; 4P PALLET POSITION DOWN
      ANI     M4408  ; 4P PALLET STOPPER DOWN
      ANI     M4409  ; 4P INFRA AUTO END
      OUT     M4407  ; 4P PALLET POSITION DOWN
      AND     X536  ; INFRA 4P PALLET POSITION DOWN
      LDI     SM400  ; ALWAYS ON
      ANI     X580  ; #1 TAP LASER W/D 2P STOPPER DETE
      ANI     X583  ; #1 TAP LASER W/D 2P PLT POSI UP
      AND     X584  ; #1 TAP LASER W/D 2P PLT POSI DN
      LDI     X538  ; BUFFER STOPPER PALLET DETECT
      ANI     Y570  ; BUFFER STOPPER DOWN
      ORB
      ANB
      OUT     T4407 K20
4493  LD      M31  ; AUTO MDOE #3
      AND     T4407
      OR      M4408  ; 4P PALLET STOPPER DOWN
      ANI     M4409  ; 4P INFRA AUTO END
      OUT     M4408  ; 4P PALLET STOPPER DOWN
      ANI     X534  ; INFRA 4P PALLET DETECT
      OUT     T4408 K8
